LIN {X 0,Y 386.268,Z 340.052,A -85,B 0,C 180,E1 13716.91,E2 13716.91} C_VEL
LIN {X 0,Y 373.935,Z 326.395,A -85,B 0,C 180,E1 13713.839,E2 13713.839} C_VEL
LIN {X 0,Y 356.934,Z 301.733,A -85,B 0,C 180,E1 13708.485,E2 13708.485} C_VEL
LIN {X 0,Y 348.808,Z 290.548,A -85,B 0,C 180,E1 13705.376,E2 13705.376} C_VEL
LIN {X 0,Y 345.384,Z 285.946,A -85,B 0,C 180,E1 13703.91,E2 13703.91} C_VEL
LIN {X 0,Y 341.987,Z 281.466,A -85,B 0,C 180,E1 13702.339,E2 13702.339} C_VEL
LIN {X 0,Y 338.204,Z 276.56,A -85,B 0,C 180,E1 13700.418,E2 13700.418} C_VEL
LIN {X 0,Y 334.673,Z 272.149,A -85,B 0,C 180,E1 13698.418,E2 13698.418} C_VEL
LIN {X 0,Y 333.52,Z 270.824,A -85,B 0,C 180,E1 13697.716,E2 13697.716} C_VEL
LIN {X 0,Y 330.176,Z 266.785,A -85,B 0,C 180,E1 13695.456,E2 13695.456} C_VEL
LIN {X 0,Y 329.315,Z 265.342,A -85,B 0,C 180,E1 13694.776,E2 13694.776} C_VEL
LIN {X 0,Y 326.007,Z 262.321,A -85,B 0,C 180,E1 13692.038,E2 13692.038} C_VEL
LIN {X 0,Y 324.468,Z 259.24,A -85,B 0,C 180,E1 13690.296,E2 13690.296} C_VEL
LIN {X 0,Y 319.963,Z 254.972,A -85,B 0,C 180,E1 13681.074,E2 13681.074} C_VEL
LIN {X 0,Y 320.128,Z 255.393,A -85,B 0,C 180,E1 13677.852,E2 13677.852} C_VEL
LIN {X 0,Y 324.571,Z 259.436,A -85,B 0,C 180,E1 13669.886,E2 13669.886} C_VEL
LIN {X 0,Y 326.879,Z 263.417,A -85,B 0,C 180,E1 13667.456,E2 13667.456} C_VEL
LIN {X 0,Y 329.69,Z 265.855,A -85,B 0,C 180,E1 13665.241,E2 13665.241} C_VEL
LIN {X 0,Y 332.506,Z 269.885,A -85,B 0,C 180,E1 13663.221,E2 13663.221} C_VEL
LIN {X 0,Y 334.533,Z 271.893,A -85,B 0,C 180,E1 13661.98,E2 13661.98} C_VEL
LIN {X 0,Y 337.954,Z 276.34,A -85,B 0,C 180,E1 13660.018,E2 13660.018} C_VEL
LIN {X 0,Y 339.714,Z 278.629,A -85,B 0,C 180,E1 13659.091,E2 13659.091} C_VEL
LIN {X 0,Y 343.732,Z 283.696,A -85,B 0,C 180,E1 13657.148,E2 13657.148} C_VEL
LIN {X 0,Y 348.055,Z 289.495,A -85,B 0,C 180,E1 13655.247,E2 13655.247} C_VEL
LIN {X 0,Y 354.37,Z 298.173,A -85,B 0,C 180,E1 13652.754,E2 13652.754} C_VEL
LIN {X 0,Y 356.73,Z 301.564,A -85,B 0,C 180,E1 13651.89,E2 13651.89} C_VEL
LIN {X 0,Y 358.866,Z 306.87,A -85,B 0,C 180,E1 13651.048,E2 13651.048} C_VEL
LIN {X 0,Y 363.911,Z 325.647,A -85,B 0,C 180,E1 13648.944,E2 13648.944} C_VEL
LIN {X 0,Y 365.246,Z 328.766,A -85,B 0,C 180,E1 13648.485,E2 13648.485} C_VEL
LIN {X 0,Y 373.121,Z 344.861,A -85,B 0,C 180,E1 13646.031,E2 13646.031} C_VEL
LIN {X 0,Y 375.226,Z 349.974,A -85,B 0,C 180,E1 13645.391,E2 13645.391} C_VEL
LIN {X 0,Y 363.631,Z 518.512,A -85,B 0,C 180,E1 13642.347,E2 13642.347} C_VEL
LIN {X 0,Y 361.378,Z 537.609,A -85,B 0,C 180,E1 13641.872,E2 13641.872} C_VEL
LIN {X 0,Y 357.513,Z 560.275,A -85,B 0,C 180,E1 13641.106,E2 13641.106} C_VEL
LIN {X 0,Y 353.084,Z 580.15,A -85,B 0,C 180,E1 13640.185,E2 13640.185} C_VEL
LIN {X 0,Y 348.65,Z 597.084,A -85,B 0,C 180,E1 13639.202,E2 13639.202} C_VEL
LIN {X 0,Y 343.899,Z 612.945,A -85,B 0,C 180,E1 13638.092,E2 13638.092} C_VEL
LIN {X 0,Y 338.731,Z 628.386,A -85,B 0,C 180,E1 13636.804,E2 13636.804} C_VEL
LIN {X 0,Y 333.209,Z 643.365,A -85,B 0,C 180,E1 13635.324,E2 13635.324} C_VEL
LIN {X 0,Y 326.894,Z 659.095,A -85,B 0,C 180,E1 13633.482,E2 13633.482} C_VEL
LIN {X 0,Y 318.806,Z 677.555,A -85,B 0,C 180,E1 13630.832,E2 13630.832} C_VEL
LIN {X 0,Y 312.71,Z 690.554,A -85,B 0,C 180,E1 13628.567,E2 13628.567} C_VEL
LIN {X 0,Y 306.921,Z 702.441,A -85,B 0,C 180,E1 13626.127,E2 13626.127} C_VEL
LIN {X 0,Y 301.69,Z 712.936,A -85,B 0,C 180,E1 13623.601,E2 13623.601} C_VEL
LIN {X 0,Y 296.723,Z 722.827,A -85,B 0,C 180,E1 13620.806,E2 13620.806} C_VEL
LIN {X 0,Y 292.163,Z 732.011,A -85,B 0,C 180,E1 13617.735,E2 13617.735} C_VEL
LIN {X 0,Y 287.756,Z 741.331,A -85,B 0,C 180,E1 13613.985,E2 13613.985} C_VEL
LIN {X 0,Y 283.988,Z 749.983,A -85,B 0,C 180,E1 13609.538,E2 13609.538} C_VEL
LIN {X 0,Y 281.915,Z 755.6,A -85,B 0,C 180,E1 13605.847,E2 13605.847} C_VEL
LIN {X 0,Y 280.717,Z 759.775,A -85,B 0,C 180,E1 13602.338,E2 13602.338} C_VEL
LIN {X 0,Y 280.122,Z 762.882,A -85,B 0,C 180,E1 13598.828,E2 13598.828} C_VEL
LIN {X 0,Y 279.95,Z 764.861,A -85,B 0,C 180,E1 13595.533,E2 13595.533} C_VEL
LIN {X 0,Y 279.965,Z 765.937,A -85,B 0,C 180,E1 13592.251,E2 13592.251} C_VEL
LIN {X 0,Y 279.98,Z 766.115,A -85,B 0,C 180,E1 13588.977,E2 13588.977} C_VEL
LIN {X 0,Y 279.944,Z 765.306,A -85,B 0,C 180,E1 13585.494,E2 13585.494} C_VEL
LIN {X 0,Y 280.051,Z 763.477,A -85,B 0,C 180,E1 13581.997,E2 13581.997} C_VEL
LIN {X 0,Y 280.571,Z 760.402,A -85,B 0,C 180,E1 13578.281,E2 13578.281} C_VEL
LIN {X 0,Y 281.653,Z 756.413,A -85,B 0,C 180,E1 13574.771,E2 13574.771} C_VEL
LIN {X 0,Y 283.447,Z 751.32,A -85,B 0,C 180,E1 13571.279,E2 13571.279} C_VEL
LIN {X 0,Y 286.041,Z 745.066,A -85,B 0,C 180,E1 13567.823,E2 13567.823} C_VEL
LIN {X 0,Y 289.479,Z 737.579,A -85,B 0,C 180,E1 13564.424,E2 13564.424} C_VEL
LIN {X 0,Y 294.639,Z 727.132,A -85,B 0,C 180,E1 13560.528,E2 13560.528} C_VEL
LIN {X 0,Y 300.694,Z 714.948,A -85,B 0,C 180,E1 13556.927,E2 13556.927} C_VEL
LIN {X 0,Y 306.139,Z 704.024,A -85,B 0,C 180,E1 13554.228,E2 13554.228} C_VEL
LIN {X 0,Y 311.866,Z 692.294,A -85,B 0,C 180,E1 13551.768,E2 13551.768} C_VEL
LIN {X 0,Y 317.867,Z 679.553,A -85,B 0,C 180,E1 13549.497,E2 13549.497} C_VEL
LIN {X 0,Y 324.119,Z 665.583,A -85,B 0,C 180,E1 13547.386,E2 13547.386} C_VEL
LIN {X 0,Y 331.869,Z 646.919,A -85,B 0,C 180,E1 13545.055,E2 13545.055} C_VEL
LIN {X 0,Y 338.168,Z 629.997,A -85,B 0,C 180,E1 13543.342,E2 13543.342} C_VEL
LIN {X 0,Y 343.312,Z 614.785,A -85,B 0,C 180,E1 13542.048,E2 13542.048} C_VEL
LIN {X 0,Y 348.21,Z 598.635,A -85,B 0,C 180,E1 13540.898,E2 13540.898} C_VEL
LIN {X 0,Y 352.296,Z 583.32,A -85,B 0,C 180,E1 13539.985,E2 13539.985} C_VEL
LIN {X 0,Y 356.088,Z 566.94,A -85,B 0,C 180,E1 13539.183,E2 13539.183} C_VEL
LIN {X 0,Y 359.407,Z 549.856,A -85,B 0,C 180,E1 13538.516,E2 13538.516} C_VEL
LIN {X 0,Y 362.097,Z 532.301,A -85,B 0,C 180,E1 13537.984,E2 13537.984} C_VEL
LIN {X 0,Y 364.159,Z 512.509,A -85,B 0,C 180,E1 13537.527,E2 13537.527} C_VEL
LIN {X 0,Y 375.197,Z 349.477,A -85,B 0,C 180,E1 13534.586,E2 13534.586} C_VEL
LIN {X 0,Y 367.633,Z 333.537,A -85,B 0,C 180,E1 13532.283,E2 13532.283} C_VEL
LIN {X 0,Y 360.351,Z 319.565,A -85,B 0,C 180,E1 13529.873,E2 13529.873} C_VEL
LIN {X 0,Y 353.374,Z 307.386,A -85,B 0,C 180,E1 13527.332,E2 13527.332} C_VEL
LIN {X 0,Y 346.425,Z 297.518,A -85,B 0,C 180,E1 13524.559,E2 13524.559} C_VEL
LIN {X 0,Y 342.821,Z 292.619,A -85,B 0,C 180,E1 13522.961,E2 13522.961} C_VEL
LIN {X 0,Y 339.925,Z 288.734,A -85,B 0,C 180,E1 13521.573,E2 13521.573} C_VEL
LIN {X 0,Y 336.229,Z 283.884,A -85,B 0,C 180,E1 13519.636,E2 13519.636} C_VEL
LIN {X 0,Y 332.684,Z 279.147,A -85,B 0,C 180,E1 13517.536,E2 13517.536} C_VEL
LIN {X 0,Y 328.89,Z 274.782,A -85,B 0,C 180,E1 13514.976,E2 13514.976} C_VEL
LIN {X 0,Y 327.794,Z 273.016,A -85,B 0,C 180,E1 13514.098,E2 13514.098} C_VEL
LIN {X 0,Y 324.631,Z 269.906,A -85,B 0,C 180,E1 13511.369,E2 13511.369} C_VEL
LIN {X 0,Y 323.127,Z 267.059,A -85,B 0,C 180,E1 13509.619,E2 13509.619} C_VEL
LIN {X 0,Y 318.996,Z 262.945,A -85,B 0,C 180,E1 13500.898,E2 13500.898} C_VEL
LIN {X 0,Y 319.101,Z 263.237,A -85,B 0,C 180,E1 13497.845,E2 13497.845} C_VEL
LIN {X 0,Y 323.392,Z 267.413,A -85,B 0,C 180,E1 13489.759,E2 13489.759} C_VEL
LIN {X 0,Y 325.671,Z 271.291,A -85,B 0,C 180,E1 13487.319,E2 13487.319} C_VEL
LIN {X 0,Y 328.214,Z 273.554,A -85,B 0,C 180,E1 13485.263,E2 13485.263} C_VEL
LIN {X 0,Y 331.228,Z 277.785,A -85,B 0,C 180,E1 13483.064,E2 13483.064} C_VEL
LIN {X 0,Y 332.948,Z 279.629,A -85,B 0,C 180,E1 13481.981,E2 13481.981} C_VEL
LIN {X 0,Y 336.629,Z 284.252,A -85,B 0,C 180,E1 13479.845,E2 13479.845} C_VEL
LIN {X 0,Y 341.914,Z 291.371,A -85,B 0,C 180,E1 13477.157,E2 13477.157} C_VEL
LIN {X 0,Y 346.173,Z 297.193,A -85,B 0,C 180,E1 13475.24,E2 13475.24} C_VEL
LIN {X 0,Y 352.796,Z 306.559,A -85,B 0,C 180,E1 13472.577,E2 13472.577} C_VEL
LIN {X 0,Y 360.002,Z 317.337,A -85,B 0,C 180,E1 13470.004,E2 13470.004} C_VEL
LIN {X 0,Y 371.633,Z 334.055,A -85,B 0,C 180,E1 13466.433,E2 13466.433} C_VEL
LIN {X 0,Y 387.013,Z 350.884,A -85,B 0,C 180,E1 13462.616,E2 13462.616} C_VEL
LIN {X 0,Y 404.416,Z 365.915,A -85,B 0,C 180,E1 13459.019,E2 13459.019} C_VEL
LIN {X 0,Y 413.951,Z 373.978,A -85,B 0,C 180,E1 13456.97,E2 13456.97} C_VEL
LIN {X 0,Y 423.451,Z 382.101,A -85,B 0,C 180,E1 13454.752,E2 13454.752} C_VEL
LIN {X 0,Y 431.998,Z 389.621,A -85,B 0,C 180,E1 13452.556,E2 13452.556} C_VEL
LIN {X 0,Y 441.62,Z 398.394,A -85,B 0,C 180,E1 13449.815,E2 13449.815} C_VEL
LIN {X 0,Y 450.481,Z 406.222,A -85,B 0,C 180,E1 13447.171,E2 13447.171} C_VEL
LIN {X 0,Y 459.526,Z 414.01,A -85,B 0,C 180,E1 13444.334,E2 13444.334} C_VEL
LIN {X 0,Y 466.257,Z 419.625,A -85,B 0,C 180,E1 13442.104,E2 13442.104} C_VEL
LIN {X 0,Y 473.318,Z 425.906,A -85,B 0,C 180,E1 13439.621,E2 13439.621} C_VEL
LIN {X 0,Y 478.445,Z 429.943,A -85,B 0,C 180,E1 13437.74,E2 13437.74} C_VEL
LIN {X 0,Y 484.241,Z 434.888,A -85,B 0,C 180,E1 13435.432,E2 13435.432} C_VEL
LIN {X 0,Y 488.516,Z 438.069,A -85,B 0,C 180,E1 13433.648,E2 13433.648} C_VEL
LIN {X 0,Y 493.363,Z 442.438,A -85,B 0,C 180,E1 13431.392,E2 13431.392} C_VEL
LIN {X 0,Y 498.263,Z 445.648,A -85,B 0,C 180,E1 13428.969,E2 13428.969} C_VEL
LIN {X 0,Y 502.59,Z 449.801,A -85,B 0,C 180,E1 13426.478,E2 13426.478} C_VEL
LIN {X 0,Y 506.276,Z 452.541,A -85,B 0,C 180,E1 13424.057,E2 13424.057} C_VEL
LIN {X 0,Y 509.659,Z 454.3,A -85,B 0,C 180,E1 13421.542,E2 13421.542} C_VEL
LIN {X 0,Y 510.793,Z 455.335,A -85,B 0,C 180,E1 13420.488,E2 13420.488} C_VEL
LIN {X 0,Y 513.093,Z 457.868,A -85,B 0,C 180,E1 13417.952,E2 13417.952} C_VEL
LIN {X 0,Y 514.62,Z 459.31,A -85,B 0,C 180,E1 13415.686,E2 13415.686} C_VEL
LIN {X 0,Y 515.845,Z 460.261,A -85,B 0,C 180,E1 13413,E2 13413} C_VEL
LIN {X 0,Y 516.274,Z 460.529,A -85,B 0,C 180,E1 13410.555,E2 13410.555} C_VEL
LIN {X 0,Y 516.046,Z 460.366,A -85,B 0,C 180,E1 13407.779,E2 13407.779} C_VEL
LIN {X 0,Y 515.181,Z 459.728,A -85,B 0,C 180,E1 13405.325,E2 13405.325} C_VEL
LIN {X 0,Y 513.6,Z 458.417,A -85,B 0,C 180,E1 13402.731,E2 13402.731} C_VEL
LIN {X 0,Y 511.457,Z 456.139,A -85,B 0,C 180,E1 13400.169,E2 13400.169} C_VEL
LIN {X 0,Y 509.789,Z 454.349,A -85,B 0,C 180,E1 13398.576,E2 13398.576} C_VEL
LIN {X 0,Y 506.453,Z 452.644,A -85,B 0,C 180,E1 13396.064,E2 13396.064} C_VEL
LIN {X 0,Y 502.909,Z 450.074,A -85,B 0,C 180,E1 13393.722,E2 13393.722} C_VEL
LIN {X 0,Y 498.849,Z 446.206,A -85,B 0,C 180,E1 13391.358,E2 13391.358} C_VEL
LIN {X 0,Y 493.606,Z 442.619,A -85,B 0,C 180,E1 13388.72,E2 13388.72} C_VEL
LIN {X 0,Y 488.817,Z 438.383,A -85,B 0,C 180,E1 13386.495,E2 13386.495} C_VEL
LIN {X 0,Y 485.363,Z 435.679,A -85,B 0,C 180,E1 13385.018,E2 13385.018} C_VEL
LIN {X 0,Y 479.539,Z 431.003,A -85,B 0,C 180,E1 13382.699,E2 13382.699} C_VEL
LIN {X 0,Y 475.675,Z 427.655,A -85,B 0,C 180,E1 13381.23,E2 13381.23} C_VEL
LIN {X 0,Y 469.252,Z 422.415,A -85,B 0,C 180,E1 13378.936,E2 13378.936} C_VEL
LIN {X 0,Y 464.33,Z 418.154,A -85,B 0,C 180,E1 13377.248,E2 13377.248} C_VEL
LIN {X 0,Y 456.023,Z 410.909,A -85,B 0,C 180,E1 13374.544,E2 13374.544} C_VEL
LIN {X 0,Y 448.696,Z 404.527,A -85,B 0,C 180,E1 13372.288,E2 13372.288} C_VEL
LIN {X 0,Y 440.156,Z 396.98,A -85,B 0,C 180,E1 13369.755,E2 13369.755} C_VEL
LIN {X 0,Y 431.296,Z 388.943,A -85,B 0,C 180,E1 13367.251,E2 13367.251} C_VEL
LIN {X 0,Y 421.982,Z 380.697,A -85,B 0,C 180,E1 13364.872,E2 13364.872} C_VEL
LIN {X 0,Y 413.139,Z 373.258,A -85,B 0,C 180,E1 13362.85,E2 13362.85} C_VEL
LIN {X 0,Y 403.162,Z 364.77,A -85,B 0,C 180,E1 13360.713,E2 13360.713} C_VEL
LIN {X 0,Y 385.913,Z 349.796,A -85,B 0,C 180,E1 13357.135,E2 13357.135} C_VEL
LIN {X 0,Y 371.026,Z 333.282,A -85,B 0,C 180,E1 13353.397,E2 13353.397} C_VEL
LIN {X 0,Y 359.686,Z 316.803,A -85,B 0,C 180,E1 13349.887,E2 13349.887} C_VEL
LIN {X 0,Y 351.241,Z 304.196,A -85,B 0,C 180,E1 13346.821,E2 13346.821} C_VEL
LIN {X 0,Y 343.795,Z 293.837,A -85,B 0,C 180,E1 13343.709,E2 13343.709} C_VEL
LIN {X 0,Y 339.862,Z 288.649,A -85,B 0,C 180,E1 13341.849,E2 13341.849} C_VEL
LIN {X 0,Y 336.322,Z 283.967,A -85,B 0,C 180,E1 13339.993,E2 13339.993} C_VEL
LIN {X 0,Y 332.758,Z 279.293,A -85,B 0,C 180,E1 13337.893,E2 13337.893} C_VEL
LIN {X 0,Y 328.737,Z 274.526,A -85,B 0,C 180,E1 13335.164,E2 13335.164} C_VEL
LIN {X 0,Y 327.895,Z 273.084,A -85,B 0,C 180,E1 13334.481,E2 13334.481} C_VEL
LIN {X 0,Y 324.677,Z 270.01,A -85,B 0,C 180,E1 13331.727,E2 13331.727} C_VEL
LIN {X 0,Y 323.175,Z 267.07,A -85,B 0,C 180,E1 13329.978,E2 13329.978} C_VEL
LIN {X 0,Y 318.987,Z 262.924,A -85,B 0,C 180,E1 13321.078,E2 13321.078} C_VEL
LIN {X 0,Y 319.12,Z 263.29,A -85,B 0,C 180,E1 13318.025,E2 13318.025} C_VEL
LIN {X 0,Y 323.351,Z 267.336,A -85,B 0,C 180,E1 13310.118,E2 13310.118} C_VEL
LIN {X 0,Y 325.712,Z 271.322,A -85,B 0,C 180,E1 13307.591,E2 13307.591} C_VEL
LIN {X 0,Y 328.256,Z 273.631,A -85,B 0,C 180,E1 13305.536,E2 13305.536} C_VEL
LIN {X 0,Y 331.282,Z 277.826,A -85,B 0,C 180,E1 13303.337,E2 13303.337} C_VEL
LIN {X 0,Y 332.936,Z 279.602,A -85,B 0,C 180,E1 13302.297,E2 13302.297} C_VEL
LIN {X 0,Y 336.535,Z 284.175,A -85,B 0,C 180,E1 13300.202,E2 13300.202} C_VEL
LIN {X 0,Y 341.897,Z 291.332,A -85,B 0,C 180,E1 13297.473,E2 13297.473} C_VEL
LIN {X 0,Y 346.064,Z 297.019,A -85,B 0,C 180,E1 13295.595,E2 13295.595} C_VEL
LIN {X 0,Y 352.278,Z 305.799,A -85,B 0,C 180,E1 13293.082,E2 13293.082} C_VEL
LIN {X 0,Y 355.942,Z 311.724,A -85,B 0,C 180,E1 13291.703,E2 13291.703} C_VEL
LIN {X 0,Y 362.038,Z 322.693,A -85,B 0,C 180,E1 13289.549,E2 13289.549} C_VEL
LIN {X 0,Y 365.246,Z 328.766,A -85,B 0,C 180,E1 13288.485,E2 13288.485} C_VEL
LIN {X 0,Y 366.5,Z 332.86,A -85,B 0,C 180,E1 13288.021,E2 13288.021} C_VEL
LIN {X 0,Y 368.162,Z 346.842,A -85,B 0,C 180,E1 13287.118,E2 13287.118} C_VEL
LIN {X 0,Y 369.102,Z 349.82,A -85,B 0,C 180,E1 13286.791,E2 13286.791} C_VEL
LIN {X 0,Y 370.477,Z 353.325,A -85,B 0,C 180,E1 13286.35,E2 13286.35} C_VEL
LIN {X 0,Y 358.789,Z 518.345,A -85,B 0,C 180,E1 13283.361,E2 13283.361} C_VEL
LIN {X 0,Y 356.461,Z 537.596,A -85,B 0,C 180,E1 13282.882,E2 13282.882} C_VEL
LIN {X 0,Y 352.312,Z 561.069,A -85,B 0,C 180,E1 13282.081,E2 13282.081} C_VEL
LIN {X 0,Y 347.999,Z 579.939,A -85,B 0,C 180,E1 13281.203,E2 13281.203} C_VEL
LIN {X 0,Y 343.442,Z 596.908,A -85,B 0,C 180,E1 13280.219,E2 13280.219} C_VEL
LIN {X 0,Y 338.565,Z 612.769,A -85,B 0,C 180,E1 13279.108,E2 13279.108} C_VEL
LIN {X 0,Y 333.249,Z 628.209,A -85,B 0,C 180,E1 13277.817,E2 13277.817} C_VEL
LIN {X 0,Y 327.566,Z 643.188,A -85,B 0,C 180,E1 13276.331,E2 13276.331} C_VEL
LIN {X 0,Y 321.054,Z 658.917,A -85,B 0,C 180,E1 13274.479,E2 13274.479} C_VEL
LIN {X 0,Y 312.923,Z 676.917,A -85,B 0,C 180,E1 13271.882,E2 13271.882} C_VEL
LIN {X 0,Y 306.383,Z 690.376,A -85,B 0,C 180,E1 13269.516,E2 13269.516} C_VEL
LIN {X 0,Y 300.369,Z 702.263,A -85,B 0,C 180,E1 13267.045,E2 13267.045} C_VEL
LIN {X 0,Y 294.917,Z 712.758,A -85,B 0,C 180,E1 13264.48,E2 13264.48} C_VEL
LIN {X 0,Y 289.728,Z 722.649,A -85,B 0,C 180,E1 13261.635,E2 13261.635} C_VEL
LIN {X 0,Y 284.949,Z 731.833,A -85,B 0,C 180,E1 13258.5,E2 13258.5} C_VEL
LIN {X 0,Y 280.306,Z 741.152,A -85,B 0,C 180,E1 13254.664,E2 13254.664} C_VEL
LIN {X 0,Y 276.312,Z 749.804,A -85,B 0,C 180,E1 13250.104,E2 13250.104} C_VEL
LIN {X 0,Y 274.095,Z 755.423,A -85,B 0,C 180,E1 13246.311,E2 13246.311} C_VEL
LIN {X 0,Y 272.799,Z 759.597,A -85,B 0,C 180,E1 13242.702,E2 13242.702} C_VEL
LIN {X 0,Y 272.148,Z 762.705,A -85,B 0,C 180,E1 13239.089,E2 13239.089} C_VEL
LIN {X 0,Y 271.955,Z 764.686,A -85,B 0,C 180,E1 13235.696,E2 13235.696} C_VEL
LIN {X 0,Y 271.965,Z 765.762,A -85,B 0,C 180,E1 13232.317,E2 13232.317} C_VEL
LIN {X 0,Y 271.981,Z 765.94,A -85,B 0,C 180,E1 13228.947,E2 13228.947} C_VEL
LIN {X 0,Y 271.944,Z 765.131,A -85,B 0,C 180,E1 13225.361,E2 13225.361} C_VEL
LIN {X 0,Y 272.082,Z 763.152,A -85,B 0,C 180,E1 13221.548,E2 13221.548} C_VEL
LIN {X 0,Y 272.642,Z 760.225,A -85,B 0,C 180,E1 13217.935,E2 13217.935} C_VEL
LIN {X 0,Y 273.813,Z 756.235,A -85,B 0,C 180,E1 13214.324,E2 13214.324} C_VEL
LIN {X 0,Y 275.735,Z 751.141,A -85,B 0,C 180,E1 13210.735,E2 13210.735} C_VEL
LIN {X 0,Y 278.49,Z 744.888,A -85,B 0,C 180,E1 13207.188,E2 13207.188} C_VEL
LIN {X 0,Y 282.123,Z 737.4,A -85,B 0,C 180,E1 13203.707,E2 13203.707} C_VEL
LIN {X 0,Y 287.548,Z 726.954,A -85,B 0,C 180,E1 13199.726,E2 13199.726} C_VEL
LIN {X 0,Y 293.83,Z 714.862,A -85,B 0,C 180,E1 13196.082,E2 13196.082} C_VEL
LIN {X 0,Y 299.554,Z 703.846,A -85,B 0,C 180,E1 13193.316,E2 13193.316} C_VEL
LIN {X 0,Y 305.486,Z 692.155,A -85,B 0,C 180,E1 13190.83,E2 13190.83} C_VEL
LIN {X 0,Y 311.725,Z 679.375,A -85,B 0,C 180,E1 13188.526,E2 13188.526} C_VEL
LIN {X 0,Y 318.191,Z 665.406,A -85,B 0,C 180,E1 13186.396,E2 13186.396} C_VEL
LIN {X 0,Y 326.187,Z 646.742,A -85,B 0,C 180,E1 13184.05,E2 13184.05} C_VEL
LIN {X 0,Y 332.77,Z 629.544,A -85,B 0,C 180,E1 13182.304,E2 13182.304} C_VEL
LIN {X 0,Y 338.263,Z 613.689,A -85,B 0,C 180,E1 13180.962,E2 13180.962} C_VEL
LIN {X 0,Y 343.101,Z 598.075,A -85,B 0,C 180,E1 13179.856,E2 13179.856} C_VEL
LIN {X 0,Y 347.497,Z 581.901,A -85,B 0,C 180,E1 13178.901,E2 13178.901} C_VEL
LIN {X 0,Y 351.332,Z 565.526,A -85,B 0,C 180,E1 13178.112,E2 13178.112} C_VEL
LIN {X 0,Y 354.815,Z 547.736,A -85,B 0,C 180,E1 13177.434,E2 13177.434} C_VEL
LIN {X 0,Y 358.133,Z 525.425,A -85,B 0,C 180,E1 13176.79,E2 13176.79} C_VEL
LIN {X 0,Y 360.831,Z 491.406,A -85,B 0,C 180,E1 13176.123,E2 13176.123} C_VEL
LIN {X 0,Y 370.425,Z 352.817,A -85,B 0,C 180,E1 13173.621,E2 13173.621} C_VEL
LIN {X 0,Y 363.461,Z 337.977,A -85,B 0,C 180,E1 13171.398,E2 13171.398} C_VEL
LIN {X 0,Y 355.897,Z 323.266,A -85,B 0,C 180,E1 13168.759,E2 13168.759} C_VEL
LIN {X 0,Y 350.2,Z 313.406,A -85,B 0,C 180,E1 13166.587,E2 13166.587} C_VEL
LIN {X 0,Y 343.823,Z 304.159,A -85,B 0,C 180,E1 13163.934,E2 13163.934} C_VEL
LIN {X 0,Y 338.469,Z 296.639,A -85,B 0,C 180,E1 13161.398,E2 13161.398} C_VEL
LIN {X 0,Y 334.22,Z 291.13,A -85,B 0,C 180,E1 13159.123,E2 13159.123} C_VEL
LIN {X 0,Y 330.453,Z 286.11,A -85,B 0,C 180,E1 13156.796,E2 13156.796} C_VEL
LIN {X 0,Y 327.14,Z 281.961,A -85,B 0,C 180,E1 13154.424,E2 13154.424} C_VEL
LIN {X 0,Y 326.197,Z 280.616,A -85,B 0,C 180,E1 13153.652,E2 13153.652} C_VEL
LIN {X 0,Y 323.15,Z 277.325,A -85,B 0,C 180,E1 13150.88,E2 13150.88} C_VEL
LIN {X 0,Y 321.846,Z 274.873,A -85,B 0,C 180,E1 13149.297,E2 13149.297} C_VEL
LIN {X 0,Y 318.008,Z 270.854,A -85,B 0,C 180,E1 13140.721,E2 13140.721} C_VEL
LIN {X 0,Y 318.154,Z 271.253,A -85,B 0,C 180,E1 13137.659,E2 13137.659} C_VEL
LIN {X 0,Y 322.179,Z 275.301,A -85,B 0,C 180,E1 13129.991,E2 13129.991} C_VEL
LIN {X 0,Y 324.508,Z 279.194,A -85,B 0,C 180,E1 13127.454,E2 13127.454} C_VEL
LIN {X 0,Y 326.793,Z 281.317,A -85,B 0,C 180,E1 13125.56,E2 13125.56} C_VEL
LIN {X 0,Y 330.007,Z 285.727,A -85,B 0,C 180,E1 13123.181,E2 13123.181} C_VEL
LIN {X 0,Y 331.427,Z 287.428,A -85,B 0,C 180,E1 13122.259,E2 13122.259} C_VEL
LIN {X 0,Y 335.791,Z 293.151,A -85,B 0,C 180,E1 13119.694,E2 13119.694} C_VEL
LIN {X 0,Y 339.93,Z 298.753,A -85,B 0,C 180,E1 13117.564,E2 13117.564} C_VEL
LIN {X 0,Y 345.555,Z 306.5,A -85,B 0,C 180,E1 13115.01,E2 13115.01} C_VEL
LIN {X 0,Y 354.41,Z 319.625,A -85,B 0,C 180,E1 13111.524,E2 13111.524} C_VEL
LIN {X 0,Y 368.498,Z 340.631,A -85,B 0,C 180,E1 13106.948,E2 13106.948} C_VEL
LIN {X 0,Y 383.658,Z 357.495,A -85,B 0,C 180,E1 13103.078,E2 13103.078} C_VEL
LIN {X 0,Y 403.445,Z 374.675,A -85,B 0,C 180,E1 13098.946,E2 13098.946} C_VEL
LIN {X 0,Y 411.876,Z 381.715,A -85,B 0,C 180,E1 13097.143,E2 13097.143} C_VEL
LIN {X 0,Y 421.313,Z 389.639,A -85,B 0,C 180,E1 13094.989,E2 13094.989} C_VEL
LIN {X 0,Y 429.934,Z 397.176,A -85,B 0,C 180,E1 13092.788,E2 13092.788} C_VEL
LIN {X 0,Y 438.951,Z 405.269,A -85,B 0,C 180,E1 13090.262,E2 13090.262} C_VEL
LIN {X 0,Y 448.23,Z 413.453,A -85,B 0,C 180,E1 13087.511,E2 13087.511} C_VEL
LIN {X 0,Y 457.07,Z 420.986,A -85,B 0,C 180,E1 13084.77,E2 13084.77} C_VEL
LIN {X 0,Y 464.208,Z 427.004,A -85,B 0,C 180,E1 13082.43,E2 13082.43} C_VEL
LIN {X 0,Y 471.575,Z 433.471,A -85,B 0,C 180,E1 13079.863,E2 13079.863} C_VEL
LIN {X 0,Y 476.902,Z 437.655,A -85,B 0,C 180,E1 13077.919,E2 13077.919} C_VEL
LIN {X 0,Y 482.84,Z 442.669,A -85,B 0,C 180,E1 13075.576,E2 13075.576} C_VEL
LIN {X 0,Y 487.337,Z 446.052,A -85,B 0,C 180,E1 13073.709,E2 13073.709} C_VEL
LIN {X 0,Y 492.23,Z 450.378,A -85,B 0,C 180,E1 13071.444,E2 13071.444} C_VEL
LIN {X 0,Y 497.637,Z 454.079,A -85,B 0,C 180,E1 13068.75,E2 13068.75} C_VEL
LIN {X 0,Y 501.65,Z 457.858,A -85,B 0,C 180,E1 13066.439,E2 13066.439} C_VEL
LIN {X 0,Y 505.24,Z 460.477,A -85,B 0,C 180,E1 13064.087,E2 13064.087} C_VEL
LIN {X 0,Y 508.651,Z 462.234,A -85,B 0,C 180,E1 13061.565,E2 13061.565} C_VEL
LIN {X 0,Y 509.906,Z 463.464,A -85,B 0,C 180,E1 13060.392,E2 13060.392} C_VEL
LIN {X 0,Y 512.177,Z 465.921,A -85,B 0,C 180,E1 13057.853,E2 13057.853} C_VEL
LIN {X 0,Y 513.706,Z 467.304,A -85,B 0,C 180,E1 13055.584,E2 13055.584} C_VEL
LIN {X 0,Y 514.89,Z 468.216,A -85,B 0,C 180,E1 13052.894,E2 13052.894} C_VEL
LIN {X 0,Y 515.314,Z 468.47,A -85,B 0,C 180,E1 13050.445,E2 13050.445} C_VEL
LIN {X 0,Y 515.067,Z 468.307,A -85,B 0,C 180,E1 13047.775,E2 13047.775} C_VEL
LIN {X 0,Y 514.243,Z 467.711,A -85,B 0,C 180,E1 13045.428,E2 13045.428} C_VEL
LIN {X 0,Y 512.605,Z 466.365,A -85,B 0,C 180,E1 13042.717,E2 13042.717} C_VEL
LIN {X 0,Y 510.459,Z 464.113,A -85,B 0,C 180,E1 13040.158,E2 13040.158} C_VEL
LIN {X 0,Y 508.78,Z 462.283,A -85,B 0,C 180,E1 13038.553,E2 13038.553} C_VEL
LIN {X 0,Y 505.417,Z 460.579,A -85,B 0,C 180,E1 13036.035,E2 13036.035} C_VEL
LIN {X 0,Y 501.851,Z 458.028,A -85,B 0,C 180,E1 13033.687,E2 13033.687} C_VEL
LIN {X 0,Y 497.753,Z 454.206,A -85,B 0,C 180,E1 13031.315,E2 13031.315} C_VEL
LIN {X 0,Y 492.529,Z 450.598,A -85,B 0,C 180,E1 13028.695,E2 13028.695} C_VEL
LIN {X 0,Y 487.641,Z 446.35,A -85,B 0,C 180,E1 13026.428,E2 13026.428} C_VEL
LIN {X 0,Y 484.306,Z 443.686,A -85,B 0,C 180,E1 13025.006,E2 13025.006} C_VEL
LIN {X 0,Y 478.388,Z 439.045,A -85,B 0,C 180,E1 13022.661,E2 13022.661} C_VEL
LIN {X 0,Y 473.956,Z 435.228,A -85,B 0,C 180,E1 13020.977,E2 13020.977} C_VEL
LIN {X 0,Y 467.477,Z 429.951,A -85,B 0,C 180,E1 13018.689,E2 13018.689} C_VEL
LIN {X 0,Y 461.873,Z 425.194,A -85,B 0,C 180,E1 13016.795,E2 13016.795} C_VEL
LIN {X 0,Y 453.321,Z 417.813,A -85,B 0,C 180,E1 13014.047,E2 13014.047} C_VEL
LIN {X 0,Y 446.033,Z 411.325,A -85,B 0,C 180,E1 13011.817,E2 13011.817} C_VEL
LIN {X 0,Y 438.152,Z 404.504,A -85,B 0,C 180,E1 13009.508,E2 13009.508} C_VEL
LIN {X 0,Y 429.304,Z 396.593,A -85,B 0,C 180,E1 13007.048,E2 13007.048} C_VEL
LIN {X 0,Y 419.866,Z 388.363,A -85,B 0,C 180,E1 13004.678,E2 13004.678} C_VEL
LIN {X 0,Y 411.376,Z 381.28,A -85,B 0,C 180,E1 13002.746,E2 13002.746} C_VEL
LIN {X 0,Y 401.592,Z 373.078,A -85,B 0,C 180,E1 13000.671,E2 13000.671} C_VEL
LIN {X 0,Y 382.303,Z 356.118,A -85,B 0,C 180,E1 12996.607,E2 12996.607} C_VEL
LIN {X 0,Y 367.9,Z 339.853,A -85,B 0,C 180,E1 12992.88,E2 12992.88} C_VEL
LIN {X 0,Y 351.607,Z 315.368,A -85,B 0,C 180,E1 12987.432,E2 12987.432} C_VEL
LIN {X 0,Y 343.843,Z 304.211,A -85,B 0,C 180,E1 12984.252,E2 12984.252} C_VEL
LIN {X 0,Y 338.408,Z 296.559,A -85,B 0,C 180,E1 12981.675,E2 12981.675} C_VEL
LIN {X 0,Y 334.311,Z 291.217,A -85,B 0,C 180,E1 12979.48,E2 12979.48} C_VEL
LIN {X 0,Y 330.398,Z 286.089,A -85,B 0,C 180,E1 12977.071,E2 12977.071} C_VEL
LIN {X 0,Y 326.995,Z 281.702,A -85,B 0,C 180,E1 12974.612,E2 12974.612} C_VEL
LIN {X 0,Y 326.262,Z 280.671,A -85,B 0,C 180,E1 12974.011,E2 12974.011} C_VEL
LIN {X 0,Y 323.194,Z 277.434,A -85,B 0,C 180,E1 12971.239,E2 12971.239} C_VEL
LIN {X 0,Y 321.892,Z 274.896,A -85,B 0,C 180,E1 12969.656,E2 12969.656} C_VEL
LIN {X 0,Y 318.002,Z 270.826,A -85,B 0,C 180,E1 12960.901,E2 12960.901} C_VEL
LIN {X 0,Y 318.209,Z 271.374,A -85,B 0,C 180,E1 12957.659,E2 12957.659} C_VEL
LIN {X 0,Y 322.139,Z 275.22,A -85,B 0,C 180,E1 12950.351,E2 12950.351} C_VEL
LIN {X 0,Y 324.548,Z 279.224,A -85,B 0,C 180,E1 12947.726,E2 12947.726} C_VEL
LIN {X 0,Y 326.773,Z 281.271,A -85,B 0,C 180,E1 12945.885,E2 12945.885} C_VEL
LIN {X 0,Y 329.803,Z 285.514,A -85,B 0,C 180,E1 12943.623,E2 12943.623} C_VEL
LIN {X 0,Y 331.352,Z 287.293,A -85,B 0,C 180,E1 12942.618,E2 12942.618} C_VEL
LIN {X 0,Y 335.757,Z 293.139,A -85,B 0,C 180,E1 12940.018,E2 12940.018} C_VEL
LIN {X 0,Y 339.911,Z 298.713,A -85,B 0,C 180,E1 12937.881,E2 12937.881} C_VEL
LIN {X 0,Y 345.624,Z 306.575,A -85,B 0,C 180,E1 12935.289,E2 12935.289} C_VEL
LIN {X 0,Y 351.746,Z 315.892,A -85,B 0,C 180,E1 12932.809,E2 12932.809} C_VEL
LIN {X 0,Y 358.447,Z 328.069,A -85,B 0,C 180,E1 12930.321,E2 12930.321} C_VEL
LIN {X 0,Y 366.358,Z 343.88,A -85,B 0,C 180,E1 12927.66,E2 12927.66} C_VEL
LIN {X 0,Y 369.102,Z 349.82,A -85,B 0,C 180,E1 12926.791,E2 12926.791} C_VEL
LIN {X 0,Y 369.576,Z 352.536,A -85,B 0,C 180,E1 12926.586,E2 12926.586} C_VEL
LIN {X 0,Y 369.012,Z 357.168,A -85,B 0,C 180,E1 12926.558,E2 12926.558} C_VEL
LIN {X 0,Y 365.102,Z 370.077,A -85,B 0,C 180,E1 12927.035,E2 12927.035} C_VEL
LIN {X 0,Y 364.616,Z 373.344,A -85,B 0,C 180,E1 12927.037,E2 12927.037} C_VEL
LIN {X 0,Y 354.042,Z 518.375,A -85,B 0,C 180,E1 12924.398,E2 12924.398} C_VEL
LIN {X 0,Y 351.612,Z 537.907,A -85,B 0,C 180,E1 12923.91,E2 12923.91} C_VEL
LIN {X 0,Y 347.267,Z 561.637,A -85,B 0,C 180,E1 12923.094,E2 12923.094} C_VEL
LIN {X 0,Y 342.829,Z 580.482,A -85,B 0,C 180,E1 12922.212,E2 12922.212} C_VEL
LIN {X 0,Y 338.346,Z 596.732,A -85,B 0,C 180,E1 12921.267,E2 12921.267} C_VEL
LIN {X 0,Y 333.341,Z 612.593,A -85,B 0,C 180,E1 12920.156,E2 12920.156} C_VEL
LIN {X 0,Y 327.876,Z 628.033,A -85,B 0,C 180,E1 12918.864,E2 12918.864} C_VEL
LIN {X 0,Y 322.028,Z 643.011,A -85,B 0,C 180,E1 12917.373,E2 12917.373} C_VEL
LIN {X 0,Y 315.278,Z 658.825,A -85,B 0,C 180,E1 12915.501,E2 12915.501} C_VEL
LIN {X 0,Y 306.636,Z 677.295,A -85,B 0,C 180,E1 12912.803,E2 12912.803} C_VEL
LIN {X 0,Y 300.144,Z 690.198,A -85,B 0,C 180,E1 12910.506,E2 12910.506} C_VEL
LIN {X 0,Y 293.899,Z 702.085,A -85,B 0,C 180,E1 12908.003,E2 12908.003} C_VEL
LIN {X 0,Y 288.16,Z 712.689,A -85,B 0,C 180,E1 12905.37,E2 12905.37} C_VEL
LIN {X 0,Y 282.799,Z 722.47,A -85,B 0,C 180,E1 12902.504,E2 12902.504} C_VEL
LIN {X 0,Y 277.788,Z 731.654,A -85,B 0,C 180,E1 12899.305,E2 12899.305} C_VEL
LIN {X 0,Y 272.896,Z 740.974,A -85,B 0,C 180,E1 12895.381,E2 12895.381} C_VEL
LIN {X 0,Y 268.661,Z 749.626,A -85,B 0,C 180,E1 12890.703,E2 12890.703} C_VEL
LIN {X 0,Y 266.26,Z 755.321,A -85,B 0,C 180,E1 12886.742,E2 12886.742} C_VEL
LIN {X 0,Y 264.888,Z 759.42,A -85,B 0,C 180,E1 12883.088,E2 12883.088} C_VEL
LIN {X 0,Y 264.172,Z 762.529,A -85,B 0,C 180,E1 12879.365,E2 12879.365} C_VEL
LIN {X 0,Y 263.961,Z 764.51,A -85,B 0,C 180,E1 12875.869,E2 12875.869} C_VEL
LIN {X 0,Y 263.965,Z 765.587,A -85,B 0,C 180,E1 12872.388,E2 12872.388} C_VEL
LIN {X 0,Y 263.982,Z 765.765,A -85,B 0,C 180,E1 12868.915,E2 12868.915} C_VEL
LIN {X 0,Y 263.944,Z 764.9,A -85,B 0,C 180,E1 12865.084,E2 12865.084} C_VEL
LIN {X 0,Y 264.106,Z 762.975,A -85,B 0,C 180,E1 12861.291,E2 12861.291} C_VEL
LIN {X 0,Y 264.719,Z 760.048,A -85,B 0,C 180,E1 12857.569,E2 12857.569} C_VEL
LIN {X 0,Y 265.987,Z 756.057,A -85,B 0,C 180,E1 12853.851,E2 12853.851} C_VEL
LIN {X 0,Y 268.049,Z 750.963,A -85,B 0,C 180,E1 12850.159,E2 12850.159} C_VEL
LIN {X 0,Y 270.975,Z 744.709,A -85,B 0,C 180,E1 12846.518,E2 12846.518} C_VEL
LIN {X 0,Y 274.815,Z 737.222,A -85,B 0,C 180,E1 12842.952,E2 12842.952} C_VEL
LIN {X 0,Y 280.516,Z 726.775,A -85,B 0,C 180,E1 12838.884,E2 12838.884} C_VEL
LIN {X 0,Y 287.083,Z 714.684,A -85,B 0,C 180,E1 12835.172,E2 12835.172} C_VEL
LIN {X 0,Y 293.204,Z 703.379,A -85,B 0,C 180,E1 12832.296,E2 12832.296} C_VEL
LIN {X 0,Y 299.213,Z 691.977,A -85,B 0,C 180,E1 12829.844,E2 12829.844} C_VEL
LIN {X 0,Y 305.678,Z 679.197,A -85,B 0,C 180,E1 12827.516,E2 12827.516} C_VEL
LIN {X 0,Y 312.259,Z 665.443,A -85,B 0,C 180,E1 12825.4,E2 12825.4} C_VEL
LIN {X 0,Y 320.327,Z 647.275,A -85,B 0,C 180,E1 12823.087,E2 12823.087} C_VEL
LIN {X 0,Y 327.282,Z 629.644,A -85,B 0,C 180,E1 12821.283,E2 12821.283} C_VEL
LIN {X 0,Y 332.723,Z 614.433,A -85,B 0,C 180,E1 12819.985,E2 12819.985} C_VEL
LIN {X 0,Y 337.711,Z 598.855,A -85,B 0,C 180,E1 12818.869,E2 12818.869} C_VEL
LIN {X 0,Y 342.18,Z 582.969,A -85,B 0,C 180,E1 12817.92,E2 12817.92} C_VEL
LIN {X 0,Y 346.267,Z 566.094,A -85,B 0,C 180,E1 12817.099,E2 12817.099} C_VEL
LIN {X 0,Y 349.765,Z 548.819,A -85,B 0,C 180,E1 12816.434,E2 12816.434} C_VEL
LIN {X 0,Y 352.683,Z 530.329,A -85,B 0,C 180,E1 12815.885,E2 12815.885} C_VEL
LIN {X 0,Y 355.148,Z 505.654,A -85,B 0,C 180,E1 12815.343,E2 12815.343} C_VEL
LIN {X 0,Y 365.762,Z 356.152,A -85,B 0,C 180,E1 12812.631,E2 12812.631} C_VEL
LIN {X 0,Y 358.297,Z 340.185,A -85,B 0,C 180,E1 12810.112,E2 12810.112} C_VEL
LIN {X 0,Y 351.653,Z 327.366,A -85,B 0,C 180,E1 12807.658,E2 12807.658} C_VEL
LIN {X 0,Y 347.377,Z 319.846,A -85,B 0,C 180,E1 12805.946,E2 12805.946} C_VEL
LIN {X 0,Y 340.095,Z 308.94,A -85,B 0,C 180,E1 12802.744,E2 12802.744} C_VEL
LIN {X 0,Y 335.591,Z 302.895,A -85,B 0,C 180,E1 12800.493,E2 12800.493} C_VEL
LIN {X 0,Y 332.382,Z 298.52,A -85,B 0,C 180,E1 12798.686,E2 12798.686} C_VEL
LIN {X 0,Y 328.713,Z 293.564,A -85,B 0,C 180,E1 12796.342,E2 12796.342} C_VEL
LIN {X 0,Y 325.492,Z 289.268,A -85,B 0,C 180,E1 12793.928,E2 12793.928} C_VEL
LIN {X 0,Y 324.589,Z 288.186,A -85,B 0,C 180,E1 12793.177,E2 12793.177} C_VEL
LIN {X 0,Y 321.694,Z 284.735,A -85,B 0,C 180,E1 12790.386,E2 12790.386} C_VEL
LIN {X 0,Y 320.728,Z 282.759,A -85,B 0,C 180,E1 12789.149,E2 12789.149} C_VEL
LIN {X 0,Y 317.033,Z 278.802,A -85,B 0,C 180,E1 12780.723,E2 12780.723} C_VEL
LIN {X 0,Y 317.151,Z 279.15,A -85,B 0,C 180,E1 12777.823,E2 12777.823} C_VEL
LIN {X 0,Y 320.973,Z 283.18,A -85,B 0,C 180,E1 12770.225,E2 12770.225} C_VEL
LIN {X 0,Y 323.254,Z 286.994,A -85,B 0,C 180,E1 12767.677,E2 12767.677} C_VEL
LIN {X 0,Y 325.382,Z 289.066,A -85,B 0,C 180,E1 12765.859,E2 12765.859} C_VEL
LIN {X 0,Y 328.661,Z 293.54,A -85,B 0,C 180,E1 12763.383,E2 12763.383} C_VEL
LIN {X 0,Y 330.168,Z 295.616,A -85,B 0,C 180,E1 12762.372,E2 12762.372} C_VEL
LIN {X 0,Y 333.977,Z 300.614,A -85,B 0,C 180,E1 12760.089,E2 12760.089} C_VEL
LIN {X 0,Y 338.044,Z 306.249,A -85,B 0,C 180,E1 12757.935,E2 12757.935} C_VEL
LIN {X 0,Y 343.472,Z 313.966,A -85,B 0,C 180,E1 12755.399,E2 12755.399} C_VEL
LIN {X 0,Y 351.481,Z 326.072,A -85,B 0,C 180,E1 12752.144,E2 12752.144} C_VEL
LIN {X 0,Y 365.747,Z 347.666,A -85,B 0,C 180,E1 12747.367,E2 12747.367} C_VEL
LIN {X 0,Y 381.003,Z 364.781,A -85,B 0,C 180,E1 12743.388,E2 12743.388} C_VEL
LIN {X 0,Y 402.341,Z 383.247,A -85,B 0,C 180,E1 12738.903,E2 12738.903} C_VEL
LIN {X 0,Y 411.923,Z 391.196,A -85,B 0,C 180,E1 12736.85,E2 12736.85} C_VEL
LIN {X 0,Y 420.903,Z 398.719,A -85,B 0,C 180,E1 12734.789,E2 12734.789} C_VEL
LIN {X 0,Y 430.119,Z 406.715,A -85,B 0,C 180,E1 12732.431,E2 12732.431} C_VEL
LIN {X 0,Y 437.632,Z 413.425,A -85,B 0,C 180,E1 12730.311,E2 12730.311} C_VEL
LIN {X 0,Y 446.468,Z 421.137,A -85,B 0,C 180,E1 12727.704,E2 12727.704} C_VEL
LIN {X 0,Y 455.709,Z 428.984,A -85,B 0,C 180,E1 12724.854,E2 12724.854} C_VEL
LIN {X 0,Y 462.919,Z 434.939,A -85,B 0,C 180,E1 12722.503,E2 12722.503} C_VEL
LIN {X 0,Y 470.055,Z 441.207,A -85,B 0,C 180,E1 12720.03,E2 12720.03} C_VEL
LIN {X 0,Y 475.413,Z 445.416,A -85,B 0,C 180,E1 12718.079,E2 12718.079} C_VEL
LIN {X 0,Y 481.431,Z 450.447,A -85,B 0,C 180,E1 12715.723,E2 12715.723} C_VEL
LIN {X 0,Y 485.976,Z 453.866,A -85,B 0,C 180,E1 12713.844,E2 12713.844} C_VEL
LIN {X 0,Y 491.103,Z 458.321,A -85,B 0,C 180,E1 12711.493,E2 12711.493} C_VEL
LIN {X 0,Y 496.542,Z 462.077,A -85,B 0,C 180,E1 12708.793,E2 12708.793} C_VEL
LIN {X 0,Y 500.593,Z 465.813,A -85,B 0,C 180,E1 12706.475,E2 12706.475} C_VEL
LIN {X 0,Y 504.204,Z 468.412,A -85,B 0,C 180,E1 12704.116,E2 12704.116} C_VEL
LIN {X 0,Y 507.498,Z 470.114,A -85,B 0,C 180,E1 12701.704,E2 12701.704} C_VEL
LIN {X 0,Y 508.661,Z 471.173,A -85,B 0,C 180,E1 12700.62,E2 12700.62} C_VEL
LIN {X 0,Y 510.947,Z 473.58,A -85,B 0,C 180,E1 12698.212,E2 12698.212} C_VEL
LIN {X 0,Y 512.581,Z 475.145,A -85,B 0,C 180,E1 12695.812,E2 12695.812} C_VEL
LIN {X 0,Y 513.83,Z 476.1,A -85,B 0,C 180,E1 12693.235,E2 12693.235} C_VEL
LIN {X 0,Y 514.295,Z 476.405,A -85,B 0,C 180,E1 12690.78,E2 12690.78} C_VEL
LIN {X 0,Y 514.203,Z 476.345,A -85,B 0,C 180,E1 12688.189,E2 12688.189} C_VEL
LIN {X 0,Y 513.349,Z 475.736,A -85,B 0,C 180,E1 12685.644,E2 12685.644} C_VEL
LIN {X 0,Y 511.883,Z 474.54,A -85,B 0,C 180,E1 12683.045,E2 12683.045} C_VEL
LIN {X 0,Y 509.79,Z 472.465,A -85,B 0,C 180,E1 12680.518,E2 12680.518} C_VEL
LIN {X 0,Y 507.643,Z 470.167,A -85,B 0,C 180,E1 12678.412,E2 12678.412} C_VEL
LIN {X 0,Y 504.38,Z 468.514,A -85,B 0,C 180,E1 12676.006,E2 12676.006} C_VEL
LIN {X 0,Y 500.793,Z 465.981,A -85,B 0,C 180,E1 12673.651,E2 12673.651} C_VEL
LIN {X 0,Y 496.657,Z 462.2,A -85,B 0,C 180,E1 12671.273,E2 12671.273} C_VEL
LIN {X 0,Y 493.397,Z 459.913,A -85,B 0,C 180,E1 12669.603,E2 12669.603} C_VEL
LIN {X 0,Y 488.21,Z 455.962,A -85,B 0,C 180,E1 12667.167,E2 12667.167} C_VEL
LIN {X 0,Y 483.536,Z 451.883,A -85,B 0,C 180,E1 12665.118,E2 12665.118} C_VEL
LIN {X 0,Y 477.635,Z 447.43,A -85,B 0,C 180,E1 12662.78,E2 12662.78} C_VEL
LIN {X 0,Y 472.433,Z 442.966,A -85,B 0,C 180,E1 12660.815,E2 12660.815} C_VEL
LIN {X 0,Y 465.973,Z 437.737,A -85,B 0,C 180,E1 12658.535,E2 12658.535} C_VEL
LIN {X 0,Y 460.328,Z 432.97,A -85,B 0,C 180,E1 12656.646,E2 12656.646} C_VEL
LIN {X 0,Y 451.498,Z 425.405,A -85,B 0,C 180,E1 12653.826,E2 12653.826} C_VEL
LIN {X 0,Y 444.007,Z 418.778,A -85,B 0,C 180,E1 12651.548,E2 12651.548} C_VEL
LIN {X 0,Y 436.148,Z 412.028,A -85,B 0,C 180,E1 12649.261,E2 12649.261} C_VEL
LIN {X 0,Y 427.346,Z 404.24,A -85,B 0,C 180,E1 12646.838,E2 12646.838} C_VEL
LIN {X 0,Y 418.408,Z 396.603,A -85,B 0,C 180,E1 12644.635,E2 12644.635} C_VEL
LIN {X 0,Y 410.162,Z 389.743,A -85,B 0,C 180,E1 12642.76,E2 12642.76} C_VEL
LIN {X 0,Y 399.145,Z 380.605,A -85,B 0,C 180,E1 12640.453,E2 12640.453} C_VEL
LIN {X 0,Y 379.125,Z 362.856,A -85,B 0,C 180,E1 12636.165,E2 12636.165} C_VEL
LIN {X 0,Y 364.806,Z 346.424,A -85,B 0,C 180,E1 12632.355,E2 12632.355} C_VEL
LIN {X 0,Y 348.941,Z 322.115,A -85,B 0,C 180,E1 12626.874,E2 12626.874} C_VEL
LIN {X 0,Y 341.284,Z 310.847,A -85,B 0,C 180,E1 12623.619,E2 12623.619} C_VEL
LIN {X 0,Y 336.002,Z 303.378,A -85,B 0,C 180,E1 12621.014,E2 12621.014} C_VEL
LIN {X 0,Y 332.472,Z 298.61,A -85,B 0,C 180,E1 12619.045,E2 12619.045} C_VEL
LIN {X 0,Y 328.766,Z 293.637,A -85,B 0,C 180,E1 12616.687,E2 12616.687} C_VEL
LIN {X 0,Y 325.481,Z 289.254,A -85,B 0,C 180,E1 12614.227,E2 12614.227} C_VEL
LIN {X 0,Y 324.442,Z 288.077,A -85,B 0,C 180,E1 12613.364,E2 12613.364} C_VEL
LIN {X 0,Y 321.588,Z 284.566,A -85,B 0,C 180,E1 12610.57,E2 12610.57} C_VEL
LIN {X 0,Y 320.773,Z 282.786,A -85,B 0,C 180,E1 12609.509,E2 12609.509} C_VEL
LIN {X 0,Y 317.026,Z 278.776,A -85,B 0,C 180,E1 12600.904,E2 12600.904} C_VEL
LIN {X 0,Y 317.199,Z 279.264,A -85,B 0,C 180,E1 12597.832,E2 12597.832} C_VEL
LIN {X 0,Y 320.933,Z 283.089,A -85,B 0,C 180,E1 12590.586,E2 12590.586} C_VEL
LIN {X 0,Y 323.386,Z 287.121,A -85,B 0,C 180,E1 12587.863,E2 12587.863} C_VEL
LIN {X 0,Y 325.323,Z 288.944,A -85,B 0,C 180,E1 12586.22,E2 12586.22} C_VEL
LIN {X 0,Y 328.458,Z 293.325,A -85,B 0,C 180,E1 12583.827,E2 12583.827} C_VEL
LIN {X 0,Y 329.841,Z 295.077,A -85,B 0,C 180,E1 12582.899,E2 12582.899} C_VEL
LIN {X 0,Y 334.027,Z 300.73,A -85,B 0,C 180,E1 12580.366,E2 12580.366} C_VEL
LIN {X 0,Y 337.944,Z 306.09,A -85,B 0,C 180,E1 12578.294,E2 12578.294} C_VEL
LIN {X 0,Y 343.451,Z 313.892,A -85,B 0,C 180,E1 12575.718,E2 12575.718} C_VEL
LIN {X 0,Y 349.074,Z 322.634,A -85,B 0,C 180,E1 12573.366,E2 12573.366} C_VEL
LIN {X 0,Y 355.471,Z 334.573,A -85,B 0,C 180,E1 12570.904,E2 12570.904} C_VEL
LIN {X 0,Y 362.883,Z 349.773,A -85,B 0,C 180,E1 12568.315,E2 12568.315} C_VEL
LIN {X 0,Y 365.834,Z 356.674,A -85,B 0,C 180,E1 12567.333,E2 12567.333} C_VEL
LIN {X 0,Y 364.616,Z 373.344,A -85,B 0,C 180,E1 12567.037,E2 12567.037} C_VEL
LIN {X 0,Y 363.511,Z 381.031,A -85,B 0,C 180,E1 12567.032,E2 12567.032} C_VEL
LIN {X 0,Y 358.613,Z 401.497,A -85,B 0,C 180,E1 12567.499,E2 12567.499} C_VEL
LIN {X 0,Y 357.722,Z 408.095,A -85,B 0,C 180,E1 12567.482,E2 12567.482} C_VEL
LIN {X 0,Y 349.415,Z 518.405,A -85,B 0,C 180,E1 12565.463,E2 12565.463} C_VEL
LIN {X 0,Y 346.824,Z 538.601,A -85,B 0,C 180,E1 12564.957,E2 12564.957} C_VEL
LIN {X 0,Y 342.334,Z 562.204,A -85,B 0,C 180,E1 12564.136,E2 12564.136} C_VEL
LIN {X 0,Y 337.963,Z 580.307,A -85,B 0,C 180,E1 12563.289,E2 12563.289} C_VEL
LIN {X 0,Y 333.366,Z 596.556,A -85,B 0,C 180,E1 12562.347,E2 12562.347} C_VEL
LIN {X 0,Y 328.231,Z 612.417,A -85,B 0,C 180,E1 12561.237,E2 12561.237} C_VEL
LIN {X 0,Y 322.617,Z 627.856,A -85,B 0,C 180,E1 12559.945,E2 12559.945} C_VEL
LIN {X 0,Y 316.6,Z 642.834,A -85,B 0,C 180,E1 12558.451,E2 12558.451} C_VEL
LIN {X 0,Y 309.682,Z 658.563,A -85,B 0,C 180,E1 12556.583,E2 12556.583} C_VEL
LIN {X 0,Y 300.77,Z 677.022,A -85,B 0,C 180,E1 12553.872,E2 12553.872} C_VEL
LIN {X 0,Y 293.999,Z 690.02,A -85,B 0,C 180,E1 12551.537,E2 12551.537} C_VEL
LIN {X 0,Y 287.514,Z 701.906,A -85,B 0,C 180,E1 12549.004,E2 12549.004} C_VEL
LIN {X 0,Y 281.603,Z 712.401,A -85,B 0,C 180,E1 12546.362,E2 12546.362} C_VEL
LIN {X 0,Y 275.938,Z 722.291,A -85,B 0,C 180,E1 12543.416,E2 12543.416} C_VEL
LIN {X 0,Y 270.684,Z 731.475,A -85,B 0,C 180,E1 12540.153,E2 12540.153} C_VEL
LIN {X 0,Y 265.531,Z 740.795,A -85,B 0,C 180,E1 12536.137,E2 12536.137} C_VEL
LIN {X 0,Y 261.04,Z 749.447,A -85,B 0,C 180,E1 12531.336,E2 12531.336} C_VEL
LIN {X 0,Y 258.503,Z 755.067,A -85,B 0,C 180,E1 12527.325,E2 12527.325} C_VEL
LIN {X 0,Y 256.957,Z 759.345,A -85,B 0,C 180,E1 12523.388,E2 12523.388} C_VEL
LIN {X 0,Y 256.202,Z 762.352,A -85,B 0,C 180,E1 12519.66,E2 12519.66} C_VEL
LIN {X 0,Y 255.966,Z 764.334,A -85,B 0,C 180,E1 12516.053,E2 12516.053} C_VEL
LIN {X 0,Y 255.965,Z 765.412,A -85,B 0,C 180,E1 12512.462,E2 12512.462} C_VEL
LIN {X 0,Y 255.983,Z 765.591,A -85,B 0,C 180,E1 12508.881,E2 12508.881} C_VEL
LIN {X 0,Y 255.944,Z 764.756,A -85,B 0,C 180,E1 12505.009,E2 12505.009} C_VEL
LIN {X 0,Y 256.136,Z 762.779,A -85,B 0,C 180,E1 12500.987,E2 12500.987} C_VEL
LIN {X 0,Y 256.806,Z 759.871,A -85,B 0,C 180,E1 12497.179,E2 12497.179} C_VEL
LIN {X 0,Y 258.178,Z 755.879,A -85,B 0,C 180,E1 12493.348,E2 12493.348} C_VEL
LIN {X 0,Y 260.392,Z 750.778,A -85,B 0,C 180,E1 12489.546,E2 12489.546} C_VEL
LIN {X 0,Y 263.5,Z 744.531,A -85,B 0,C 180,E1 12485.81,E2 12485.81} C_VEL
LIN {X 0,Y 267.555,Z 737.043,A -85,B 0,C 180,E1 12482.155,E2 12482.155} C_VEL
LIN {X 0,Y 273.549,Z 726.593,A -85,B 0,C 180,E1 12477.997,E2 12477.997} C_VEL
LIN {X 0,Y 280.413,Z 714.505,A -85,B 0,C 180,E1 12474.218,E2 12474.218} C_VEL
LIN {X 0,Y 286.632,Z 703.489,A -85,B 0,C 180,E1 12471.366,E2 12471.366} C_VEL
LIN {X 0,Y 293.035,Z 691.799,A -85,B 0,C 180,E1 12468.817,E2 12468.817} C_VEL
LIN {X 0,Y 299.473,Z 679.519,A -85,B 0,C 180,E1 12466.551,E2 12466.551} C_VEL
LIN {X 0,Y 306.088,Z 666.172,A -85,B 0,C 180,E1 12464.466,E2 12464.466} C_VEL
LIN {X 0,Y 313.683,Z 649.742,A -85,B 0,C 180,E1 12462.318,E2 12462.318} C_VEL
LIN {X 0,Y 321.688,Z 630.314,A -85,B 0,C 180,E1 12460.28,E2 12460.28} C_VEL
LIN {X 0,Y 327.598,Z 614.256,A -85,B 0,C 180,E1 12458.904,E2 12458.904} C_VEL
LIN {X 0,Y 332.716,Z 598.679,A -85,B 0,C 180,E1 12457.789,E2 12457.789} C_VEL
LIN {X 0,Y 337.296,Z 582.793,A -85,B 0,C 180,E1 12456.843,E2 12456.843} C_VEL
LIN {X 0,Y 341.482,Z 565.918,A -85,B 0,C 180,E1 12456.024,E2 12456.024} C_VEL
LIN {X 0,Y 345.082,Z 548.529,A -85,B 0,C 180,E1 12455.358,E2 12455.358} C_VEL
LIN {X 0,Y 348.087,Z 529.859,A -85,B 0,C 180,E1 12454.808,E2 12454.808} C_VEL
LIN {X 0,Y 350.69,Z 503.823,A -85,B 0,C 180,E1 12454.244,E2 12454.244} C_VEL
LIN {X 0,Y 361.247,Z 359.755,A -85,B 0,C 180,E1 12451.636,E2 12451.636} C_VEL
LIN {X 0,Y 354.224,Z 344.497,A -85,B 0,C 180,E1 12449.139,E2 12449.139} C_VEL
LIN {X 0,Y 347.831,Z 331.91,A -85,B 0,C 180,E1 12446.644,E2 12446.644} C_VEL
LIN {X 0,Y 343.788,Z 324.944,A -85,B 0,C 180,E1 12444.944,E2 12444.944} C_VEL
LIN {X 0,Y 337.191,Z 315.153,A -85,B 0,C 180,E1 12441.894,E2 12441.894} C_VEL
LIN {X 0,Y 333.546,Z 310.063,A -85,B 0,C 180,E1 12439.983,E2 12439.983} C_VEL
LIN {X 0,Y 330.564,Z 305.905,A -85,B 0,C 180,E1 12438.244,E2 12438.244} C_VEL
LIN {X 0,Y 327.118,Z 301.132,A -85,B 0,C 180,E1 12435.968,E2 12435.968} C_VEL
LIN {X 0,Y 323.923,Z 296.684,A -85,B 0,C 180,E1 12433.477,E2 12433.477} C_VEL
LIN {X 0,Y 320.334,Z 292.284,A -85,B 0,C 180,E1 12429.976,E2 12429.976} C_VEL
LIN {X 0,Y 319.463,Z 290.565,A -85,B 0,C 180,E1 12428.822,E2 12428.822} C_VEL
LIN {X 0,Y 316.046,Z 286.726,A -85,B 0,C 180,E1 12420.544,E2 12420.544} C_VEL
LIN {X 0,Y 316.2,Z 287.186,A -85,B 0,C 180,E1 12417.644,E2 12417.644} C_VEL
LIN {X 0,Y 319.711,Z 290.889,A -85,B 0,C 180,E1 12410.55,E2 12410.55} C_VEL
LIN {X 0,Y 322.097,Z 294.892,A -85,B 0,C 180,E1 12407.814,E2 12407.814} C_VEL
LIN {X 0,Y 323.982,Z 296.806,A -85,B 0,C 180,E1 12406.162,E2 12406.162} C_VEL
LIN {X 0,Y 327.445,Z 301.47,A -85,B 0,C 180,E1 12403.502,E2 12403.502} C_VEL
LIN {X 0,Y 332.332,Z 308.313,A -85,B 0,C 180,E1 12400.399,E2 12400.399} C_VEL
LIN {X 0,Y 336.251,Z 313.856,A -85,B 0,C 180,E1 12398.271,E2 12398.271} C_VEL
LIN {X 0,Y 341.321,Z 321.277,A -85,B 0,C 180,E1 12395.833,E2 12395.833} C_VEL
LIN {X 0,Y 349.074,Z 333.247,A -85,B 0,C 180,E1 12392.588,E2 12392.588} C_VEL
LIN {X 0,Y 362.55,Z 354.088,A -85,B 0,C 180,E1 12387.933,E2 12387.933} C_VEL
LIN {X 0,Y 377.425,Z 371.119,A -85,B 0,C 180,E1 12383.928,E2 12383.928} C_VEL
LIN {X 0,Y 399.496,Z 390.404,A -85,B 0,C 180,E1 12379.213,E2 12379.213} C_VEL
LIN {X 0,Y 409.871,Z 398.905,A -85,B 0,C 180,E1 12377.021,E2 12377.021} C_VEL
LIN {X 0,Y 416.859,Z 404.724,A -85,B 0,C 180,E1 12375.435,E2 12375.435} C_VEL
LIN {X 0,Y 425.864,Z 412.324,A -85,B 0,C 180,E1 12373.244,E2 12373.244} C_VEL
LIN {X 0,Y 434.702,Z 420.094,A -85,B 0,C 180,E1 12370.821,E2 12370.821} C_VEL
LIN {X 0,Y 444.28,Z 428.426,A -85,B 0,C 180,E1 12368.028,E2 12368.028} C_VEL
LIN {X 0,Y 453.465,Z 436.17,A -85,B 0,C 180,E1 12365.219,E2 12365.219} C_VEL
LIN {X 0,Y 460.836,Z 442.287,A -85,B 0,C 180,E1 12362.844,E2 12362.844} C_VEL
LIN {X 0,Y 468.405,Z 448.836,A -85,B 0,C 180,E1 12360.246,E2 12360.246} C_VEL
LIN {X 0,Y 473.885,Z 453.146,A -85,B 0,C 180,E1 12358.252,E2 12358.252} C_VEL
LIN {X 0,Y 480.039,Z 458.235,A -85,B 0,C 180,E1 12355.864,E2 12355.864} C_VEL
LIN {X 0,Y 484.444,Z 461.517,A -85,B 0,C 180,E1 12354.053,E2 12354.053} C_VEL
LIN {X 0,Y 489.67,Z 466.034,A -85,B 0,C 180,E1 12351.688,E2 12351.688} C_VEL
LIN {X 0,Y 494.754,Z 469.305,A -85,B 0,C 180,E1 12349.231,E2 12349.231} C_VEL
LIN {X 0,Y 498.854,Z 473.233,A -85,B 0,C 180,E1 12346.894,E2 12346.894} C_VEL
LIN {X 0,Y 502.825,Z 476.136,A -85,B 0,C 180,E1 12344.391,E2 12344.391} C_VEL
LIN {X 0,Y 506.143,Z 477.92,A -85,B 0,C 180,E1 12341.97,E2 12341.97} C_VEL
LIN {X 0,Y 507.369,Z 478.806,A -85,B 0,C 180,E1 12340.904,E2 12340.904} C_VEL
LIN {X 0,Y 509.661,Z 481.231,A -85,B 0,C 180,E1 12338.574,E2 12338.574} C_VEL
LIN {X 0,Y 511.455,Z 482.974,A -85,B 0,C 180,E1 12336.059,E2 12336.059} C_VEL
LIN {X 0,Y 512.737,Z 483.956,A -85,B 0,C 180,E1 12333.577,E2 12333.577} C_VEL
LIN {X 0,Y 513.299,Z 484.342,A -85,B 0,C 180,E1 12331.004,E2 12331.004} C_VEL
LIN {X 0,Y 513.285,Z 484.33,A -85,B 0,C 180,E1 12328.549,E2 12328.549} C_VEL
LIN {X 0,Y 512.513,Z 483.805,A -85,B 0,C 180,E1 12325.973,E2 12325.973} C_VEL
LIN {X 0,Y 511.211,Z 482.748,A -85,B 0,C 180,E1 12323.487,E2 12323.487} C_VEL
LIN {X 0,Y 509.206,Z 480.839,A -85,B 0,C 180,E1 12320.963,E2 12320.963} C_VEL
LIN {X 0,Y 507.133,Z 478.486,A -85,B 0,C 180,E1 12318.861,E2 12318.861} C_VEL
LIN {X 0,Y 503.594,Z 476.593,A -85,B 0,C 180,E1 12316.148,E2 12316.148} C_VEL
LIN {X 0,Y 499.938,Z 474.096,A -85,B 0,C 180,E1 12313.742,E2 12313.742} C_VEL
LIN {X 0,Y 495.68,Z 470.309,A -85,B 0,C 180,E1 12311.295,E2 12311.295} C_VEL
LIN {X 0,Y 493.381,Z 468.519,A -85,B 0,C 180,E1 12310.097,E2 12310.097} C_VEL
LIN {X 0,Y 488.428,Z 465.046,A -85,B 0,C 180,E1 12307.717,E2 12307.717} C_VEL
LIN {X 0,Y 482.167,Z 459.676,A -85,B 0,C 180,E1 12304.977,E2 12304.977} C_VEL
LIN {X 0,Y 476.196,Z 455.203,A -85,B 0,C 180,E1 12302.627,E2 12302.627} C_VEL
LIN {X 0,Y 470.843,Z 450.657,A -85,B 0,C 180,E1 12300.627,E2 12300.627} C_VEL
LIN {X 0,Y 464.196,Z 445.295,A -85,B 0,C 180,E1 12298.297,E2 12298.297} C_VEL
LIN {X 0,Y 458.362,Z 440.404,A -85,B 0,C 180,E1 12296.357,E2 12296.357} C_VEL
LIN {X 0,Y 449.467,Z 432.841,A -85,B 0,C 180,E1 12293.544,E2 12293.544} C_VEL
LIN {X 0,Y 440.432,Z 425.025,A -85,B 0,C 180,E1 12290.832,E2 12290.832} C_VEL
LIN {X 0,Y 432.648,Z 418.1,A -85,B 0,C 180,E1 12288.586,E2 12288.586} C_VEL
LIN {X 0,Y 424.728,Z 411.326,A -85,B 0,C 180,E1 12286.477,E2 12286.477} C_VEL
LIN {X 0,Y 416.444,Z 404.365,A -85,B 0,C 180,E1 12284.467,E2 12284.467} C_VEL
LIN {X 0,Y 409.087,Z 398.274,A -85,B 0,C 180,E1 12282.804,E2 12282.804} C_VEL
LIN {X 0,Y 397.874,Z 389.104,A -85,B 0,C 180,E1 12280.467,E2 12280.467} C_VEL
LIN {X 0,Y 376.497,Z 370.155,A -85,B 0,C 180,E1 12275.845,E2 12275.845} C_VEL
LIN {X 0,Y 362.087,Z 353.468,A -85,B 0,C 180,E1 12271.926,E2 12271.926} C_VEL
LIN {X 0,Y 346.308,Z 328.86,A -85,B 0,C 180,E1 12266.308,E2 12266.308} C_VEL
LIN {X 0,Y 338.686,Z 317.346,A -85,B 0,C 180,E1 12262.936,E2 12262.936} C_VEL
LIN {X 0,Y 333.794,Z 310.364,A -85,B 0,C 180,E1 12260.425,E2 12260.425} C_VEL
LIN {X 0,Y 330.513,Z 305.842,A -85,B 0,C 180,E1 12258.521,E2 12258.521} C_VEL
LIN {X 0,Y 327.07,Z 301.104,A -85,B 0,C 180,E1 12256.244,E2 12256.244} C_VEL
LIN {X 0,Y 323.792,Z 296.428,A -85,B 0,C 180,E1 12253.665,E2 12253.665} C_VEL
LIN {X 0,Y 320.519,Z 292.677,A -85,B 0,C 180,E1 12250.515,E2 12250.515} C_VEL
LIN {X 0,Y 319.506,Z 290.605,A -85,B 0,C 180,E1 12249.184,E2 12249.184} C_VEL
LIN {X 0,Y 316.05,Z 286.727,A -85,B 0,C 180,E1 12240.906,E2 12240.906} C_VEL
LIN {X 0,Y 316.222,Z 287.229,A -85,B 0,C 180,E1 12237.825,E2 12237.825} C_VEL
LIN {X 0,Y 319.735,Z 290.947,A -85,B 0,C 180,E1 12230.823,E2 12230.823} C_VEL
LIN {X 0,Y 322.227,Z 295.017,A -85,B 0,C 180,E1 12228,E2 12228} C_VEL
LIN {X 0,Y 323.923,Z 296.686,A -85,B 0,C 180,E1 12226.523,E2 12226.523} C_VEL
LIN {X 0,Y 327.118,Z 301.136,A -85,B 0,C 180,E1 12224.032,E2 12224.032} C_VEL
LIN {X 0,Y 332.169,Z 308.095,A -85,B 0,C 180,E1 12220.8,E2 12220.8} C_VEL
LIN {X 0,Y 336.23,Z 313.813,A -85,B 0,C 180,E1 12218.59,E2 12218.59} C_VEL
LIN {X 0,Y 341.384,Z 321.344,A -85,B 0,C 180,E1 12216.113,E2 12216.113} C_VEL
LIN {X 0,Y 346.436,Z 329.375,A -85,B 0,C 180,E1 12213.932,E2 12213.932} C_VEL
LIN {X 0,Y 352.483,Z 340.98,A -85,B 0,C 180,E1 12211.515,E2 12211.515} C_VEL
LIN {X 0,Y 359.508,Z 355.788,A -85,B 0,C 180,E1 12208.964,E2 12208.964} C_VEL
LIN {X 0,Y 361.283,Z 360.261,A -85,B 0,C 180,E1 12208.336,E2 12208.336} C_VEL
LIN {X 0,Y 357.722,Z 408.095,A -85,B 0,C 180,E1 12207.482,E2 12207.482} C_VEL
LIN {X 0,Y 356.615,Z 415.782,A -85,B 0,C 180,E1 12207.478,E2 12207.478} C_VEL
LIN {X 0,Y 351.717,Z 436.239,A -85,B 0,C 180,E1 12207.967,E2 12207.967} C_VEL
LIN {X 0,Y 350.818,Z 442.837,A -85,B 0,C 180,E1 12207.952,E2 12207.952} C_VEL
LIN {X 0,Y 344.892,Z 518.631,A -85,B 0,C 180,E1 12206.552,E2 12206.552} C_VEL
LIN {X 0,Y 342.028,Z 540.151,A -85,B 0,C 180,E1 12206.009,E2 12206.009} C_VEL
LIN {X 0,Y 337.518,Z 562.772,A -85,B 0,C 180,E1 12205.209,E2 12205.209} C_VEL
LIN {X 0,Y 333.219,Z 580.131,A -85,B 0,C 180,E1 12204.398,E2 12204.398} C_VEL
LIN {X 0,Y 328.509,Z 596.38,A -85,B 0,C 180,E1 12203.459,E2 12203.459} C_VEL
LIN {X 0,Y 323.243,Z 612.24,A -85,B 0,C 180,E1 12202.352,E2 12202.352} C_VEL
LIN {X 0,Y 317.476,Z 627.68,A -85,B 0,C 180,E1 12201.061,E2 12201.061} C_VEL
LIN {X 0,Y 311.288,Z 642.657,A -85,B 0,C 180,E1 12199.567,E2 12199.567} C_VEL
LIN {X 0,Y 303.877,Z 659.015,A -85,B 0,C 180,E1 12197.612,E2 12197.612} C_VEL
LIN {X 0,Y 294.962,Z 676.845,A -85,B 0,C 180,E1 12194.967,E2 12194.967} C_VEL
LIN {X 0,Y 287.834,Z 690.054,A -85,B 0,C 180,E1 12192.569,E2 12192.569} C_VEL
LIN {X 0,Y 281.222,Z 701.728,A -85,B 0,C 180,E1 12190.05,E2 12190.05} C_VEL
LIN {X 0,Y 275.069,Z 712.222,A -85,B 0,C 180,E1 12187.371,E2 12187.371} C_VEL
LIN {X 0,Y 269.151,Z 722.113,A -85,B 0,C 180,E1 12184.374,E2 12184.374} C_VEL
LIN {X 0,Y 263.642,Z 731.296,A -85,B 0,C 180,E1 12181.046,E2 12181.046} C_VEL
LIN {X 0,Y 258.215,Z 740.616,A -85,B 0,C 180,E1 12176.936,E2 12176.936} C_VEL
LIN {X 0,Y 253.45,Z 749.269,A -85,B 0,C 180,E1 12172.008,E2 12172.008} C_VEL
LIN {X 0,Y 250.739,Z 754.889,A -85,B 0,C 180,E1 12167.879,E2 12167.879} C_VEL
LIN {X 0,Y 249.101,Z 759.065,A -85,B 0,C 180,E1 12163.934,E2 12163.934} C_VEL
LIN {X 0,Y 248.239,Z 762.176,A -85,B 0,C 180,E1 12159.973,E2 12159.973} C_VEL
LIN {X 0,Y 247.972,Z 764.159,A -85,B 0,C 180,E1 12156.249,E2 12156.249} C_VEL
LIN {X 0,Y 247.965,Z 765.237,A -85,B 0,C 180,E1 12152.542,E2 12152.542} C_VEL
LIN {X 0,Y 247.984,Z 765.416,A -85,B 0,C 180,E1 12148.845,E2 12148.845} C_VEL
LIN {X 0,Y 247.946,Z 764.605,A -85,B 0,C 180,E1 12144.911,E2 12144.911} C_VEL
LIN {X 0,Y 248.16,Z 762.623,A -85,B 0,C 180,E1 12140.727,E2 12140.727} C_VEL
LIN {X 0,Y 248.901,Z 759.693,A -85,B 0,C 180,E1 12136.765,E2 12136.765} C_VEL
LIN {X 0,Y 250.389,Z 755.702,A -85,B 0,C 180,E1 12132.814,E2 12132.814} C_VEL
LIN {X 0,Y 252.759,Z 750.607,A -85,B 0,C 180,E1 12128.904,E2 12128.904} C_VEL
LIN {X 0,Y 256.065,Z 744.352,A -85,B 0,C 180,E1 12125.06,E2 12125.06} C_VEL
LIN {X 0,Y 260.35,Z 736.864,A -85,B 0,C 180,E1 12121.314,E2 12121.314} C_VEL
LIN {X 0,Y 266.647,Z 726.417,A -85,B 0,C 180,E1 12117.067,E2 12117.067} C_VEL
LIN {X 0,Y 273.827,Z 714.327,A -85,B 0,C 180,E1 12113.218,E2 12113.218} C_VEL
LIN {X 0,Y 280.306,Z 703.311,A -85,B 0,C 180,E1 12110.325,E2 12110.325} C_VEL
LIN {X 0,Y 286.955,Z 691.621,A -85,B 0,C 180,E1 12107.746,E2 12107.746} C_VEL
LIN {X 0,Y 293.89,Z 678.842,A -85,B 0,C 180,E1 12105.375,E2 12105.375} C_VEL
LIN {X 0,Y 300.74,Z 665.434,A -85,B 0,C 180,E1 12103.279,E2 12103.279} C_VEL
LIN {X 0,Y 309.192,Z 647.63,A -85,B 0,C 180,E1 12100.974,E2 12100.974} C_VEL
LIN {X 0,Y 316.85,Z 629.291,A -85,B 0,C 180,E1 12099.086,E2 12099.086} C_VEL
LIN {X 0,Y 322.594,Z 614.08,A -85,B 0,C 180,E1 12097.789,E2 12097.789} C_VEL
LIN {X 0,Y 327.843,Z 598.503,A -85,B 0,C 180,E1 12096.677,E2 12096.677} C_VEL
LIN {X 0,Y 332.537,Z 582.617,A -85,B 0,C 180,E1 12095.734,E2 12095.734} C_VEL
LIN {X 0,Y 336.82,Z 565.743,A -85,B 0,C 180,E1 12094.918,E2 12094.918} C_VEL
LIN {X 0,Y 340.501,Z 548.354,A -85,B 0,C 180,E1 12094.257,E2 12094.257} C_VEL
LIN {X 0,Y 343.572,Z 529.684,A -85,B 0,C 180,E1 12093.709,E2 12093.709} C_VEL
LIN {X 0,Y 346.241,Z 503.648,A -85,B 0,C 180,E1 12093.147,E2 12093.147} C_VEL
LIN {X 0,Y 356.842,Z 363.38,A -85,B 0,C 180,E1 12090.616,E2 12090.616} C_VEL
LIN {X 0,Y 350.449,Z 349.314,A -85,B 0,C 180,E1 12088.224,E2 12088.224} C_VEL
LIN {X 0,Y 344.825,Z 337.981,A -85,B 0,C 180,E1 12085.921,E2 12085.921} C_VEL
LIN {X 0,Y 341.143,Z 331.556,A -85,B 0,C 180,E1 12084.309,E2 12084.309} C_VEL
LIN {X 0,Y 334.997,Z 322.192,A -85,B 0,C 180,E1 12081.355,E2 12081.355} C_VEL
LIN {X 0,Y 331.384,Z 317.03,A -85,B 0,C 180,E1 12079.385,E2 12079.385} C_VEL
LIN {X 0,Y 328.766,Z 313.288,A -85,B 0,C 180,E1 12077.798,E2 12077.798} C_VEL
LIN {X 0,Y 325.538,Z 308.698,A -85,B 0,C 180,E1 12075.59,E2 12075.59} C_VEL
LIN {X 0,Y 322.042,Z 303.79,A -85,B 0,C 180,E1 12072.735,E2 12072.735} C_VEL
LIN {X 0,Y 319.126,Z 300.114,A -85,B 0,C 180,E1 12069.741,E2 12069.741} C_VEL
LIN {X 0,Y 318.21,Z 298.37,A -85,B 0,C 180,E1 12068.493,E2 12068.493} C_VEL
LIN {X 0,Y 315.071,Z 294.669,A -85,B 0,C 180,E1 12060.546,E2 12060.546} C_VEL
LIN {X 0,Y 315.195,Z 295.073,A -85,B 0,C 180,E1 12057.818,E2 12057.818} C_VEL
LIN {X 0,Y 318.519,Z 298.752,A -85,B 0,C 180,E1 12050.787,E2 12050.787} C_VEL
LIN {X 0,Y 320.941,Z 302.789,A -85,B 0,C 180,E1 12047.952,E2 12047.952} C_VEL
LIN {X 0,Y 322.591,Z 304.54,A -85,B 0,C 180,E1 12046.466,E2 12046.466} C_VEL
LIN {X 0,Y 326.685,Z 310.34,A -85,B 0,C 180,E1 12043.279,E2 12043.279} C_VEL
LIN {X 0,Y 330.56,Z 315.787,A -85,B 0,C 180,E1 12040.795,E2 12040.795} C_VEL
LIN {X 0,Y 334.549,Z 321.568,A -85,B 0,C 180,E1 12038.569,E2 12038.569} C_VEL
LIN {X 0,Y 339.871,Z 329.683,A -85,B 0,C 180,E1 12035.954,E2 12035.954} C_VEL
LIN {X 0,Y 346.609,Z 340.33,A -85,B 0,C 180,E1 12033.069,E2 12033.069} C_VEL
LIN {X 0,Y 359.617,Z 360.817,A -85,B 0,C 180,E1 12028.438,E2 12028.438} C_VEL
LIN {X 0,Y 374.406,Z 377.999,A -85,B 0,C 180,E1 12024.348,E2 12024.348} C_VEL
LIN {X 0,Y 396.608,Z 397.553,A -85,B 0,C 180,E1 12019.52,E2 12019.52} C_VEL
LIN {X 0,Y 407.611,Z 406.437,A -85,B 0,C 180,E1 12017.244,E2 12017.244} C_VEL
LIN {X 0,Y 416.569,Z 413.865,A -85,B 0,C 180,E1 12015.212,E2 12015.212} C_VEL
LIN {X 0,Y 425.333,Z 421.237,A -85,B 0,C 180,E1 12013.07,E2 12013.07} C_VEL
LIN {X 0,Y 433.043,Z 427.937,A -85,B 0,C 180,E1 12010.97,E2 12010.97} C_VEL
LIN {X 0,Y 442.769,Z 436.343,A -85,B 0,C 180,E1 12008.146,E2 12008.146} C_VEL
LIN {X 0,Y 452.089,Z 444.168,A -85,B 0,C 180,E1 12005.301,E2 12005.301} C_VEL
LIN {X 0,Y 459.381,Z 450.12,A -85,B 0,C 180,E1 12002.962,E2 12002.962} C_VEL
LIN {X 0,Y 466.557,Z 456.347,A -85,B 0,C 180,E1 12000.51,E2 12000.51} C_VEL
LIN {X 0,Y 472.316,Z 460.835,A -85,B 0,C 180,E1 11998.441,E2 11998.441} C_VEL
LIN {X 0,Y 478.554,Z 465.953,A -85,B 0,C 180,E1 11996.046,E2 11996.046} C_VEL
LIN {X 0,Y 483.075,Z 469.327,A -85,B 0,C 180,E1 11994.191,E2 11994.191} C_VEL
LIN {X 0,Y 488.393,Z 473.862,A -85,B 0,C 180,E1 11991.81,E2 11991.81} C_VEL
LIN {X 0,Y 493.659,Z 477.307,A -85,B 0,C 180,E1 11989.275,E2 11989.275} C_VEL
LIN {X 0,Y 497.781,Z 481.187,A -85,B 0,C 180,E1 11986.931,E2 11986.931} C_VEL
LIN {X 0,Y 501.79,Z 484.072,A -85,B 0,C 180,E1 11984.421,E2 11984.421} C_VEL
LIN {X 0,Y 505.121,Z 485.852,A -85,B 0,C 180,E1 11981.995,E2 11981.995} C_VEL
LIN {X 0,Y 506.353,Z 486.786,A -85,B 0,C 180,E1 11980.926,E2 11980.926} C_VEL
LIN {X 0,Y 508.658,Z 489.184,A -85,B 0,C 180,E1 11978.591,E2 11978.591} C_VEL
LIN {X 0,Y 510.469,Z 490.917,A -85,B 0,C 180,E1 11976.071,E2 11976.071} C_VEL
LIN {X 0,Y 511.755,Z 491.896,A -85,B 0,C 180,E1 11973.584,E2 11973.584} C_VEL
LIN {X 0,Y 512.323,Z 492.282,A -85,B 0,C 180,E1 11971.006,E2 11971.006} C_VEL
LIN {X 0,Y 512.309,Z 492.271,A -85,B 0,C 180,E1 11968.546,E2 11968.546} C_VEL
LIN {X 0,Y 511.532,Z 491.746,A -85,B 0,C 180,E1 11965.965,E2 11965.965} C_VEL
LIN {X 0,Y 510.225,Z 490.692,A -85,B 0,C 180,E1 11963.474,E2 11963.474} C_VEL
LIN {X 0,Y 508.203,Z 488.789,A -85,B 0,C 180,E1 11960.945,E2 11960.945} C_VEL
LIN {X 0,Y 506.117,Z 486.472,A -85,B 0,C 180,E1 11958.838,E2 11958.838} C_VEL
LIN {X 0,Y 502.585,Z 484.544,A -85,B 0,C 180,E1 11956.138,E2 11956.138} C_VEL
LIN {X 0,Y 498.881,Z 482.046,A -85,B 0,C 180,E1 11953.706,E2 11953.706} C_VEL
LIN {X 0,Y 494.587,Z 478.292,A -85,B 0,C 180,E1 11951.252,E2 11951.252} C_VEL
LIN {X 0,Y 492.273,Z 476.442,A -85,B 0,C 180,E1 11950.051,E2 11950.051} C_VEL
LIN {X 0,Y 487.188,Z 472.927,A -85,B 0,C 180,E1 11947.625,E2 11947.625} C_VEL
LIN {X 0,Y 481.124,Z 467.685,A -85,B 0,C 180,E1 11944.974,E2 11944.974} C_VEL
LIN {X 0,Y 475.15,Z 463.312,A -85,B 0,C 180,E1 11942.629,E2 11942.629} C_VEL
LIN {X 0,Y 469.361,Z 458.425,A -85,B 0,C 180,E1 11940.48,E2 11940.48} C_VEL
LIN {X 0,Y 462.645,Z 453.071,A -85,B 0,C 180,E1 11938.144,E2 11938.144} C_VEL
LIN {X 0,Y 456.958,Z 448.291,A -85,B 0,C 180,E1 11936.253,E2 11936.253} C_VEL
LIN {X 0,Y 448.288,Z 440.937,A -85,B 0,C 180,E1 11933.522,E2 11933.522} C_VEL
LIN {X 0,Y 440.54,Z 434.277,A -85,B 0,C 180,E1 11931.191,E2 11931.191} C_VEL
LIN {X 0,Y 431.89,Z 426.857,A -85,B 0,C 180,E1 11928.701,E2 11928.701} C_VEL
LIN {X 0,Y 423.308,Z 419.514,A -85,B 0,C 180,E1 11926.428,E2 11926.428} C_VEL
LIN {X 0,Y 415.264,Z 412.785,A -85,B 0,C 180,E1 11924.482,E2 11924.482} C_VEL
LIN {X 0,Y 405.532,Z 404.781,A -85,B 0,C 180,E1 11922.308,E2 11922.308} C_VEL
LIN {X 0,Y 394.818,Z 396.107,A -85,B 0,C 180,E1 11920.121,E2 11920.121} C_VEL
LIN {X 0,Y 373.489,Z 377.034,A -85,B 0,C 180,E1 11915.423,E2 11915.423} C_VEL
LIN {X 0,Y 359.162,Z 360.197,A -85,B 0,C 180,E1 11911.419,E2 11911.419} C_VEL
LIN {X 0,Y 343.803,Z 335.74,A -85,B 0,C 180,E1 11905.772,E2 11905.772} C_VEL
LIN {X 0,Y 335.825,Z 323.289,A -85,B 0,C 180,E1 11902.08,E2 11902.08} C_VEL
LIN {X 0,Y 330.839,Z 316.213,A -85,B 0,C 180,E1 11899.372,E2 11899.372} C_VEL
LIN {X 0,Y 328.584,Z 313.062,A -85,B 0,C 180,E1 11897.991,E2 11897.991} C_VEL
LIN {X 0,Y 325.492,Z 308.667,A -85,B 0,C 180,E1 11895.867,E2 11895.867} C_VEL
LIN {X 0,Y 322.105,Z 303.844,A -85,B 0,C 180,E1 11893.098,E2 11893.098} C_VEL
LIN {X 0,Y 319.166,Z 300.23,A -85,B 0,C 180,E1 11890.104,E2 11890.104} C_VEL
LIN {X 0,Y 318.251,Z 298.417,A -85,B 0,C 180,E1 11888.856,E2 11888.856} C_VEL
LIN {X 0,Y 315.067,Z 294.633,A -85,B 0,C 180,E1 11880.727,E2 11880.727} C_VEL
LIN {X 0,Y 315.275,Z 295.288,A -85,B 0,C 180,E1 11877.637,E2 11877.637} C_VEL
LIN {X 0,Y 318.543,Z 298.798,A -85,B 0,C 180,E1 11871.061,E2 11871.061} C_VEL
LIN {X 0,Y 321.069,Z 302.911,A -85,B 0,C 180,E1 11868.139,E2 11868.139} C_VEL
LIN {X 0,Y 322.626,Z 304.605,A -85,B 0,C 180,E1 11866.742,E2 11866.742} C_VEL
LIN {X 0,Y 326.61,Z 310.208,A -85,B 0,C 180,E1 11863.641,E2 11863.641} C_VEL
LIN {X 0,Y 330.537,Z 315.783,A -85,B 0,C 180,E1 11861.114,E2 11861.114} C_VEL
LIN {X 0,Y 334.448,Z 321.413,A -85,B 0,C 180,E1 11858.93,E2 11858.93} C_VEL
LIN {X 0,Y 339.59,Z 329.199,A -85,B 0,C 180,E1 11856.394,E2 11856.394} C_VEL
LIN {X 0,Y 343.922,Z 336.288,A -85,B 0,C 180,E1 11854.468,E2 11854.468} C_VEL
LIN {X 0,Y 349.584,Z 347.487,A -85,B 0,C 180,E1 11852.118,E2 11852.118} C_VEL
LIN {X 0,Y 356.181,Z 361.802,A -85,B 0,C 180,E1 11849.625,E2 11849.625} C_VEL
LIN {X 0,Y 356.851,Z 363.796,A -85,B 0,C 180,E1 11849.366,E2 11849.366} C_VEL
LIN {X 0,Y 350.818,Z 442.837,A -85,B 0,C 180,E1 11847.952,E2 11847.952} C_VEL
LIN {X 0,Y 349.703,Z 450.524,A -85,B 0,C 180,E1 11847.952,E2 11847.952} C_VEL
LIN {X 0,Y 344.814,Z 470.976,A -85,B 0,C 180,E1 11848.463,E2 11848.463} C_VEL
LIN {X 0,Y 343.916,Z 477.573,A -85,B 0,C 180,E1 11848.448,E2 11848.448} C_VEL
LIN {X 0,Y 340.339,Z 520.36,A -85,B 0,C 180,E1 11847.637,E2 11847.637} C_VEL
LIN {X 0,Y 336.735,Z 544.704,A -85,B 0,C 180,E1 11846.991,E2 11846.991} C_VEL
LIN {X 0,Y 332.823,Z 563.339,A -85,B 0,C 180,E1 11846.312,E2 11846.312} C_VEL
LIN {X 0,Y 328.494,Z 580.347,A -85,B 0,C 180,E1 11845.517,E2 11845.517} C_VEL
LIN {X 0,Y 323.779,Z 596.204,A -85,B 0,C 180,E1 11844.604,E2 11844.604} C_VEL
LIN {X 0,Y 318.381,Z 612.064,A -85,B 0,C 180,E1 11843.501,E2 11843.501} C_VEL
LIN {X 0,Y 312.46,Z 627.503,A -85,B 0,C 180,E1 11842.214,E2 11842.214} C_VEL
LIN {X 0,Y 306.1,Z 642.48,A -85,B 0,C 180,E1 11840.72,E2 11840.72} C_VEL
LIN {X 0,Y 298.469,Z 658.838,A -85,B 0,C 180,E1 11838.763,E2 11838.763} C_VEL
LIN {X 0,Y 289.268,Z 676.667,A -85,B 0,C 180,E1 11836.104,E2 11836.104} C_VEL
LIN {X 0,Y 282.012,Z 689.664,A -85,B 0,C 180,E1 11833.732,E2 11833.732} C_VEL
LIN {X 0,Y 275.028,Z 701.55,A -85,B 0,C 180,E1 11831.144,E2 11831.144} C_VEL
LIN {X 0,Y 268.625,Z 712.044,A -85,B 0,C 180,E1 11828.428,E2 11828.428} C_VEL
LIN {X 0,Y 262.442,Z 721.941,A -85,B 0,C 180,E1 11825.379,E2 11825.379} C_VEL
LIN {X 0,Y 256.668,Z 731.117,A -85,B 0,C 180,E1 11821.988,E2 11821.988} C_VEL
LIN {X 0,Y 250.951,Z 740.437,A -85,B 0,C 180,E1 11817.782,E2 11817.782} C_VEL
LIN {X 0,Y 245.897,Z 749.09,A -85,B 0,C 180,E1 11812.721,E2 11812.721} C_VEL
LIN {X 0,Y 242.999,Z 754.711,A -85,B 0,C 180,E1 11808.469,E2 11808.469} C_VEL
LIN {X 0,Y 241.227,Z 758.888,A -85,B 0,C 180,E1 11804.399,E2 11804.399} C_VEL
LIN {X 0,Y 240.282,Z 761.999,A -85,B 0,C 180,E1 11800.306,E2 11800.306} C_VEL
LIN {X 0,Y 239.978,Z 763.983,A -85,B 0,C 180,E1 11796.458,E2 11796.458} C_VEL
LIN {X 0,Y 239.965,Z 765.062,A -85,B 0,C 180,E1 11792.627,E2 11792.627} C_VEL
LIN {X 0,Y 239.985,Z 765.241,A -85,B 0,C 180,E1 11788.806,E2 11788.806} C_VEL
LIN {X 0,Y 239.948,Z 764.429,A -85,B 0,C 180,E1 11784.741,E2 11784.741} C_VEL
LIN {X 0,Y 240.165,Z 762.592,A -85,B 0,C 180,E1 11780.651,E2 11780.651} C_VEL
LIN {X 0,Y 241.007,Z 759.516,A -85,B 0,C 180,E1 11776.323,E2 11776.323} C_VEL
LIN {X 0,Y 242.675,Z 755.399,A -85,B 0,C 180,E1 11772.137,E2 11772.137} C_VEL
LIN {X 0,Y 245.16,Z 750.428,A -85,B 0,C 180,E1 11768.217,E2 11768.217} C_VEL
LIN {X 0,Y 248.675,Z 744.173,A -85,B 0,C 180,E1 11764.266,E2 11764.266} C_VEL
LIN {X 0,Y 253.204,Z 736.685,A -85,B 0,C 180,E1 11760.426,E2 11760.426} C_VEL
LIN {X 0,Y 259.822,Z 726.239,A -85,B 0,C 180,E1 11756.087,E2 11756.087} C_VEL
LIN {X 0,Y 267.329,Z 714.148,A -85,B 0,C 180,E1 11752.17,E2 11752.17} C_VEL
LIN {X 0,Y 274.078,Z 703.132,A -85,B 0,C 180,E1 11749.237,E2 11749.237} C_VEL
LIN {X 0,Y 280.467,Z 692.333,A -85,B 0,C 180,E1 11746.811,E2 11746.811} C_VEL
LIN {X 0,Y 287.482,Z 679.895,A -85,B 0,C 180,E1 11744.452,E2 11744.452} C_VEL
LIN {X 0,Y 294.362,Z 666.938,A -85,B 0,C 180,E1 11742.379,E2 11742.379} C_VEL
LIN {X 0,Y 301.171,Z 653.168,A -85,B 0,C 180,E1 11740.52,E2 11740.52} C_VEL
LIN {X 0,Y 308.304,Z 637.511,A -85,B 0,C 180,E1 11738.751,E2 11738.751} C_VEL
LIN {X 0,Y 316.648,Z 616.872,A -85,B 0,C 180,E1 11736.868,E2 11736.868} C_VEL
LIN {X 0,Y 322.757,Z 599.39,A -85,B 0,C 180,E1 11735.6,E2 11735.6} C_VEL
LIN {X 0,Y 327.905,Z 582.442,A -85,B 0,C 180,E1 11734.593,E2 11734.593} C_VEL
LIN {X 0,Y 332.288,Z 565.567,A -85,B 0,C 180,E1 11733.783,E2 11733.783} C_VEL
LIN {X 0,Y 336.05,Z 548.179,A -85,B 0,C 180,E1 11733.127,E2 11733.127} C_VEL
LIN {X 0,Y 339.209,Z 529.361,A -85,B 0,C 180,E1 11732.579,E2 11732.579} C_VEL
LIN {X 0,Y 341.999,Z 502.454,A -85,B 0,C 180,E1 11732.003,E2 11732.003} C_VEL
LIN {X 0,Y 352.509,Z 366.841,A -85,B 0,C 180,E1 11729.551,E2 11729.551} C_VEL
LIN {X 0,Y 345.936,Z 352.299,A -85,B 0,C 180,E1 11726.941,E2 11726.941} C_VEL
LIN {X 0,Y 340.222,Z 340.908,A -85,B 0,C 180,E1 11724.435,E2 11724.435} C_VEL
LIN {X 0,Y 333.691,Z 330.404,A -85,B 0,C 180,E1 11721.258,E2 11721.258} C_VEL
LIN {X 0,Y 329.19,Z 323.88,A -85,B 0,C 180,E1 11718.736,E2 11718.736} C_VEL
LIN {X 0,Y 326.729,Z 320.335,A -85,B 0,C 180,E1 11717.177,E2 11717.177} C_VEL
LIN {X 0,Y 323.855,Z 316.136,A -85,B 0,C 180,E1 11715.123,E2 11715.123} C_VEL
LIN {X 0,Y 320.676,Z 311.509,A -85,B 0,C 180,E1 11712.424,E2 11712.424} C_VEL
LIN {X 0,Y 317.857,Z 307.803,A -85,B 0,C 180,E1 11709.415,E2 11709.415} C_VEL
LIN {X 0,Y 317.103,Z 306.255,A -85,B 0,C 180,E1 11708.34,E2 11708.34} C_VEL
LIN {X 0,Y 314.095,Z 302.614,A -85,B 0,C 180,E1 11700.547,E2 11700.547} C_VEL
LIN {X 0,Y 314.217,Z 303.042,A -85,B 0,C 180,E1 11697.812,E2 11697.812} C_VEL
LIN {X 0,Y 317.333,Z 306.609,A -85,B 0,C 180,E1 11691.027,E2 11691.027} C_VEL
LIN {X 0,Y 319.788,Z 310.684,A -85,B 0,C 180,E1 11688.091,E2 11688.091} C_VEL
LIN {X 0,Y 321.211,Z 312.268,A -85,B 0,C 180,E1 11686.774,E2 11686.774} C_VEL
LIN {X 0,Y 325.09,Z 317.899,A -85,B 0,C 180,E1 11683.654,E2 11683.654} C_VEL
LIN {X 0,Y 328.805,Z 323.258,A -85,B 0,C 180,E1 11681.195,E2 11681.195} C_VEL
LIN {X 0,Y 333.717,Z 330.442,A -85,B 0,C 180,E1 11678.421,E2 11678.421} C_VEL
LIN {X 0,Y 341.597,Z 343.069,A -85,B 0,C 180,E1 11674.654,E2 11674.654} C_VEL
LIN {X 0,Y 349.466,Z 356.647,A -85,B 0,C 180,E1 11671.457,E2 11671.457} C_VEL
LIN {X 0,Y 360.163,Z 371.952,A -85,B 0,C 180,E1 11667.883,E2 11667.883} C_VEL
LIN {X 0,Y 374.038,Z 387.532,A -85,B 0,C 180,E1 11664.119,E2 11664.119} C_VEL
LIN {X 0,Y 396.678,Z 406.966,A -85,B 0,C 180,E1 11659.243,E2 11659.243} C_VEL
LIN {X 0,Y 407.221,Z 415.411,A -85,B 0,C 180,E1 11657.049,E2 11657.049} C_VEL
LIN {X 0,Y 415.659,Z 422.425,A -85,B 0,C 180,E1 11655.136,E2 11655.136} C_VEL
LIN {X 0,Y 424.57,Z 429.88,A -85,B 0,C 180,E1 11652.959,E2 11652.959} C_VEL
LIN {X 0,Y 432.151,Z 436.468,A -85,B 0,C 180,E1 11650.897,E2 11650.897} C_VEL
LIN {X 0,Y 440.893,Z 443.941,A -85,B 0,C 180,E1 11648.366,E2 11648.366} C_VEL
LIN {X 0,Y 450.05,Z 451.565,A -85,B 0,C 180,E1 11645.592,E2 11645.592} C_VEL
LIN {X 0,Y 457.596,Z 457.716,A -85,B 0,C 180,E1 11643.186,E2 11643.186} C_VEL
LIN {X 0,Y 465.011,Z 464.089,A -85,B 0,C 180,E1 11640.672,E2 11640.672} C_VEL
LIN {X 0,Y 470.656,Z 468.435,A -85,B 0,C 180,E1 11638.669,E2 11638.669} C_VEL
LIN {X 0,Y 476.826,Z 473.493,A -85,B 0,C 180,E1 11636.324,E2 11636.324} C_VEL
LIN {X 0,Y 481.537,Z 476.973,A -85,B 0,C 180,E1 11634.403,E2 11634.403} C_VEL
LIN {X 0,Y 486.833,Z 481.467,A -85,B 0,C 180,E1 11632.074,E2 11632.074} C_VEL
LIN {X 0,Y 491.759,Z 484.698,A -85,B 0,C 180,E1 11629.709,E2 11629.709} C_VEL
LIN {X 0,Y 496.275,Z 488.778,A -85,B 0,C 180,E1 11627.226,E2 11627.226} C_VEL
LIN {X 0,Y 500.208,Z 491.669,A -85,B 0,C 180,E1 11624.823,E2 11624.823} C_VEL
LIN {X 0,Y 503.633,Z 493.587,A -85,B 0,C 180,E1 11622.366,E2 11622.366} C_VEL
LIN {X 0,Y 505.101,Z 494.453,A -85,B 0,C 180,E1 11621.185,E2 11621.185} C_VEL
LIN {X 0,Y 507.31,Z 496.837,A -85,B 0,C 180,E1 11618.957,E2 11618.957} C_VEL
LIN {X 0,Y 509.298,Z 498.693,A -85,B 0,C 180,E1 11616.424,E2 11616.424} C_VEL
LIN {X 0,Y 510.55,Z 499.687,A -85,B 0,C 180,E1 11614.042,E2 11614.042} C_VEL
LIN {X 0,Y 511.333,Z 500.211,A -85,B 0,C 180,E1 11611.456,E2 11611.456} C_VEL
LIN {X 0,Y 511.347,Z 500.223,A -85,B 0,C 180,E1 11608.992,E2 11608.992} C_VEL
LIN {X 0,Y 510.773,Z 499.837,A -85,B 0,C 180,E1 11606.409,E2 11606.409} C_VEL
LIN {X 0,Y 509.483,Z 498.858,A -85,B 0,C 180,E1 11603.917,E2 11603.917} C_VEL
LIN {X 0,Y 507.652,Z 497.135,A -85,B 0,C 180,E1 11601.392,E2 11601.392} C_VEL
LIN {X 0,Y 505.459,Z 494.914,A -85,B 0,C 180,E1 11599.17,E2 11599.17} C_VEL
LIN {X 0,Y 504.263,Z 493.846,A -85,B 0,C 180,E1 11598.101,E2 11598.101} C_VEL
LIN {X 0,Y 500.926,Z 492.112,A -85,B 0,C 180,E1 11595.672,E2 11595.672} C_VEL
LIN {X 0,Y 496.931,Z 489.318,A -85,B 0,C 180,E1 11593.16,E2 11593.16} C_VEL
LIN {X 0,Y 492.795,Z 485.554,A -85,B 0,C 180,E1 11590.813,E2 11590.813} C_VEL
LIN {X 0,Y 487.41,Z 481.909,A -85,B 0,C 180,E1 11588.207,E2 11588.207} C_VEL
LIN {X 0,Y 482.057,Z 477.458,A -85,B 0,C 180,E1 11585.82,E2 11585.82} C_VEL
LIN {X 0,Y 478.568,Z 474.73,A -85,B 0,C 180,E1 11584.378,E2 11584.378} C_VEL
LIN {X 0,Y 472.359,Z 469.957,A -85,B 0,C 180,E1 11581.971,E2 11581.971} C_VEL
LIN {X 0,Y 467.413,Z 465.863,A -85,B 0,C 180,E1 11580.164,E2 11580.164} C_VEL
LIN {X 0,Y 460.532,Z 460.341,A -85,B 0,C 180,E1 11577.796,E2 11577.796} C_VEL
LIN {X 0,Y 453.822,Z 454.811,A -85,B 0,C 180,E1 11575.601,E2 11575.601} C_VEL
LIN {X 0,Y 445.564,Z 447.835,A -85,B 0,C 180,E1 11573.025,E2 11573.025} C_VEL
LIN {X 0,Y 436,Z 439.684,A -85,B 0,C 180,E1 11570.199,E2 11570.199} C_VEL
LIN {X 0,Y 428.094,Z 432.714,A -85,B 0,C 180,E1 11567.966,E2 11567.966} C_VEL
LIN {X 0,Y 420.046,Z 426.058,A -85,B 0,C 180,E1 11565.914,E2 11565.914} C_VEL
LIN {X 0,Y 410.08,Z 417.819,A -85,B 0,C 180,E1 11563.585,E2 11563.585} C_VEL
LIN {X 0,Y 400.722,Z 410.321,A -85,B 0,C 180,E1 11561.585,E2 11561.585} C_VEL
LIN {X 0,Y 384.233,Z 396.846,A -85,B 0,C 180,E1 11558.221,E2 11558.221} C_VEL
LIN {X 0,Y 368.969,Z 382.205,A -85,B 0,C 180,E1 11554.593,E2 11554.593} C_VEL
LIN {X 0,Y 356.044,Z 366.611,A -85,B 0,C 180,E1 11550.832,E2 11550.832} C_VEL
LIN {X 0,Y 341.237,Z 342.484,A -85,B 0,C 180,E1 11545.189,E2 11545.189} C_VEL
LIN {X 0,Y 333.638,Z 330.338,A -85,B 0,C 180,E1 11541.538,E2 11541.538} C_VEL
LIN {X 0,Y 327.747,Z 321.55,A -85,B 0,C 180,E1 11538.13,E2 11538.13} C_VEL
LIN {X 0,Y 323.813,Z 316.098,A -85,B 0,C 180,E1 11535.4,E2 11535.4} C_VEL
LIN {X 0,Y 320.541,Z 311.398,A -85,B 0,C 180,E1 11532.613,E2 11532.613} C_VEL
LIN {X 0,Y 317.764,Z 307.641,A -85,B 0,C 180,E1 11529.6,E2 11529.6} C_VEL
LIN {X 0,Y 317.144,Z 306.304,A -85,B 0,C 180,E1 11528.704,E2 11528.704} C_VEL
LIN {X 0,Y 314.092,Z 302.582,A -85,B 0,C 180,E1 11520.73,E2 11520.73} C_VEL
LIN {X 0,Y 314.266,Z 303.171,A -85,B 0,C 180,E1 11517.812,E2 11517.812} C_VEL
LIN {X 0,Y 317.357,Z 306.645,A -85,B 0,C 180,E1 11511.302,E2 11511.302} C_VEL
LIN {X 0,Y 319.732,Z 310.613,A -85,B 0,C 180,E1 11508.454,E2 11508.454} C_VEL
LIN {X 0,Y 321.244,Z 312.332,A -85,B 0,C 180,E1 11507.05,E2 11507.05} C_VEL
LIN {X 0,Y 325.016,Z 317.768,A -85,B 0,C 180,E1 11504.017,E2 11504.017} C_VEL
LIN {X 0,Y 328.848,Z 323.358,A -85,B 0,C 180,E1 11501.473,E2 11501.473} C_VEL
LIN {X 0,Y 332.679,Z 329.006,A -85,B 0,C 180,E1 11499.273,E2 11499.273} C_VEL
LIN {X 0,Y 338.403,Z 337.954,A -85,B 0,C 180,E1 11496.399,E2 11496.399} C_VEL
LIN {X 0,Y 341.877,Z 344.045,A -85,B 0,C 180,E1 11494.815,E2 11494.815} C_VEL
LIN {X 0,Y 347.144,Z 354.909,A -85,B 0,C 180,E1 11492.558,E2 11492.558} C_VEL
LIN {X 0,Y 352.552,Z 367.136,A -85,B 0,C 180,E1 11490.425,E2 11490.425} C_VEL
LIN {X 0,Y 343.916,Z 477.573,A -85,B 0,C 180,E1 11488.448,E2 11488.448} C_VEL
LIN {X 0,Y 342.824,Z 485.26,A -85,B 0,C 180,E1 11488.45,E2 11488.45} C_VEL
LIN {X 0,Y 337.957,Z 505.707,A -85,B 0,C 180,E1 11488.981,E2 11488.981} C_VEL
LIN {X 0,Y 336.945,Z 512.289,A -85,B 0,C 180,E1 11488.959,E2 11488.959} C_VEL
LIN {X 0,Y 334.574,Z 531.693,A -85,B 0,C 180,E1 11488.511,E2 11488.511} C_VEL
LIN {X 0,Y 331.506,Z 549.148,A -85,B 0,C 180,E1 11487.995,E2 11487.995} C_VEL
LIN {X 0,Y 327.71,Z 566.136,A -85,B 0,C 180,E1 11487.352,E2 11487.352} C_VEL
LIN {X 0,Y 323.053,Z 583.51,A -85,B 0,C 180,E1 11486.514,E2 11486.514} C_VEL
LIN {X 0,Y 317.098,Z 602.399,A -85,B 0,C 180,E1 11485.375,E2 11485.375} C_VEL
LIN {X 0,Y 309.245,Z 623.298,A -85,B 0,C 180,E1 11483.765,E2 11483.765} C_VEL
LIN {X 0,Y 302.332,Z 639.461,A -85,B 0,C 180,E1 11482.216,E2 11482.216} C_VEL
LIN {X 0,Y 295.658,Z 653.621,A -85,B 0,C 180,E1 11480.593,E2 11480.593} C_VEL
LIN {X 0,Y 288.654,Z 667.321,A -85,B 0,C 180,E1 11478.727,E2 11478.727} C_VEL
LIN {X 0,Y 281.53,Z 680.278,A -85,B 0,C 180,E1 11476.63,E2 11476.63} C_VEL
LIN {X 0,Y 274.057,Z 693.045,A -85,B 0,C 180,E1 11474.168,E2 11474.168} C_VEL
LIN {X 0,Y 265.064,Z 707.656,A -85,B 0,C 180,E1 11470.731,E2 11470.731} C_VEL
LIN {X 0,Y 257.059,Z 719.899,A -85,B 0,C 180,E1 11467.072,E2 11467.072} C_VEL
LIN {X 0,Y 250.838,Z 729.314,A -85,B 0,C 180,E1 11463.642,E2 11463.642} C_VEL
LIN {X 0,Y 245.505,Z 737.445,A -85,B 0,C 180,E1 11460.058,E2 11460.058} C_VEL
LIN {X 0,Y 241.088,Z 744.395,A -85,B 0,C 180,E1 11456.341,E2 11456.341} C_VEL
LIN {X 0,Y 237.41,Z 750.584,A -85,B 0,C 180,E1 11452.272,E2 11452.272} C_VEL
LIN {X 0,Y 234.622,Z 755.888,A -85,B 0,C 180,E1 11447.866,E2 11447.866} C_VEL
LIN {X 0,Y 232.667,Z 760.776,A -85,B 0,C 180,E1 11442.406,E2 11442.406} C_VEL
LIN {X 0,Y 231.998,Z 763.628,A -85,B 0,C 180,E1 11437.179,E2 11437.179} C_VEL
LIN {X 0,Y 231.962,Z 764.857,A -85,B 0,C 180,E1 11432.965,E2 11432.965} C_VEL
LIN {X 0,Y 231.989,Z 765.095,A -85,B 0,C 180,E1 11429.012,E2 11429.012} C_VEL
LIN {X 0,Y 231.951,Z 764.254,A -85,B 0,C 180,E1 11424.559,E2 11424.559} C_VEL
LIN {X 0,Y 232.195,Z 762.418,A -85,B 0,C 180,E1 11420.333,E2 11420.333} C_VEL
LIN {X 0,Y 233.126,Z 759.339,A -85,B 0,C 180,E1 11415.851,E2 11415.851} C_VEL
LIN {X 0,Y 234.876,Z 755.346,A -85,B 0,C 180,E1 11411.64,E2 11411.64} C_VEL
LIN {X 0,Y 237.597,Z 750.25,A -85,B 0,C 180,E1 11407.486,E2 11407.486} C_VEL
LIN {X 0,Y 241.336,Z 743.995,A -85,B 0,C 180,E1 11403.423,E2 11403.423} C_VEL
LIN {X 0,Y 246.123,Z 736.506,A -85,B 0,C 180,E1 11399.486,E2 11399.486} C_VEL
LIN {X 0,Y 253.076,Z 726.06,A -85,B 0,C 180,E1 11395.054,E2 11395.054} C_VEL
LIN {X 0,Y 260.927,Z 713.97,A -85,B 0,C 180,E1 11391.07,E2 11391.07} C_VEL
LIN {X 0,Y 267.953,Z 702.954,A -85,B 0,C 180,E1 11388.098,E2 11388.098} C_VEL
LIN {X 0,Y 274.585,Z 692.155,A -85,B 0,C 180,E1 11385.648,E2 11385.648} C_VEL
LIN {X 0,Y 281.696,Z 679.984,A -85,B 0,C 180,E1 11383.318,E2 11383.318} C_VEL
LIN {X 0,Y 288.833,Z 666.985,A -85,B 0,C 180,E1 11381.223,E2 11381.223} C_VEL
LIN {X 0,Y 295.972,Z 652.991,A -85,B 0,C 180,E1 11379.328,E2 11379.328} C_VEL
LIN {X 0,Y 303.309,Z 637.33,A -85,B 0,C 180,E1 11377.559,E2 11377.559} C_VEL
LIN {X 0,Y 311.951,Z 616.489,A -85,B 0,C 180,E1 11375.666,E2 11375.666} C_VEL
LIN {X 0,Y 318.137,Z 599.213,A -85,B 0,C 180,E1 11374.42,E2 11374.42} C_VEL
LIN {X 0,Y 323.408,Z 582.266,A -85,B 0,C 180,E1 11373.42,E2 11373.42} C_VEL
LIN {X 0,Y 327.891,Z 565.392,A -85,B 0,C 180,E1 11372.616,E2 11372.616} C_VEL
LIN {X 0,Y 331.733,Z 548.003,A -85,B 0,C 180,E1 11371.966,E2 11371.966} C_VEL
LIN {X 0,Y 334.959,Z 529.186,A -85,B 0,C 180,E1 11371.423,E2 11371.423} C_VEL
LIN {X 0,Y 337.818,Z 502.278,A -85,B 0,C 180,E1 11370.85,E2 11370.85} C_VEL
LIN {X 0,Y 348.284,Z 370.452,A -85,B 0,C 180,E1 11368.462,E2 11368.462} C_VEL
LIN {X 0,Y 342.116,Z 356.552,A -85,B 0,C 180,E1 11365.862,E2 11365.862} C_VEL
LIN {X 0,Y 337.211,Z 346.761,A -85,B 0,C 180,E1 11363.597,E2 11363.597} C_VEL
LIN {X 0,Y 331.225,Z 337.026,A -85,B 0,C 180,E1 11360.544,E2 11360.544} C_VEL
LIN {X 0,Y 326.013,Z 328.999,A -85,B 0,C 180,E1 11357.4,E2 11357.4} C_VEL
LIN {X 0,Y 322.308,Z 323.695,A -85,B 0,C 180,E1 11354.737,E2 11354.737} C_VEL
LIN {X 0,Y 319.32,Z 319.225,A -85,B 0,C 180,E1 11352.111,E2 11352.111} C_VEL
LIN {X 0,Y 316.535,Z 315.353,A -85,B 0,C 180,E1 11348.996,E2 11348.996} C_VEL
LIN {X 0,Y 315.865,Z 314.06,A -85,B 0,C 180,E1 11348.007,E2 11348.007} C_VEL
LIN {X 0,Y 313.111,Z 310.543,A -85,B 0,C 180,E1 11340.366,E2 11340.366} C_VEL
LIN {X 0,Y 313.265,Z 311.105,A -85,B 0,C 180,E1 11337.622,E2 11337.622} C_VEL
LIN {X 0,Y 316.154,Z 314.459,A -85,B 0,C 180,E1 11331.268,E2 11331.268} C_VEL
LIN {X 0,Y 318.637,Z 318.578,A -85,B 0,C 180,E1 11328.231,E2 11328.231} C_VEL
LIN {X 0,Y 319.84,Z 319.993,A -85,B 0,C 180,E1 11327.084,E2 11327.084} C_VEL
LIN {X 0,Y 323.624,Z 325.65,A -85,B 0,C 180,E1 11323.947,E2 11323.947} C_VEL
LIN {X 0,Y 327.131,Z 330.835,A -85,B 0,C 180,E1 11321.558,E2 11321.558} C_VEL
LIN {X 0,Y 331.783,Z 337.861,A -85,B 0,C 180,E1 11318.845,E2 11318.845} C_VEL
LIN {X 0,Y 339.232,Z 350.116,A -85,B 0,C 180,E1 11315.164,E2 11315.164} C_VEL
LIN {X 0,Y 347.03,Z 363.898,A -85,B 0,C 180,E1 11311.895,E2 11311.895} C_VEL
LIN {X 0,Y 357.574,Z 379.109,A -85,B 0,C 180,E1 11308.284,E2 11308.284} C_VEL
LIN {X 0,Y 371.159,Z 394.548,A -85,B 0,C 180,E1 11304.511,E2 11304.511} C_VEL
LIN {X 0,Y 393.792,Z 414.119,A -85,B 0,C 180,E1 11299.553,E2 11299.553} C_VEL
LIN {X 0,Y 404.512,Z 422.603,A -85,B 0,C 180,E1 11297.368,E2 11297.368} C_VEL
LIN {X 0,Y 413.862,Z 430.265,A -85,B 0,C 180,E1 11295.267,E2 11295.267} C_VEL
LIN {X 0,Y 422.941,Z 437.792,A -85,B 0,C 180,E1 11293.07,E2 11293.07} C_VEL
LIN {X 0,Y 431.549,Z 445.205,A -85,B 0,C 180,E1 11290.742,E2 11290.742} C_VEL
LIN {X 0,Y 439.384,Z 451.862,A -85,B 0,C 180,E1 11288.479,E2 11288.479} C_VEL
LIN {X 0,Y 448.672,Z 459.553,A -85,B 0,C 180,E1 11285.678,E2 11285.678} C_VEL
LIN {X 0,Y 456.91,Z 466.217,A -85,B 0,C 180,E1 11283.055,E2 11283.055} C_VEL
LIN {X 0,Y 463.906,Z 472.165,A -85,B 0,C 180,E1 11280.684,E2 11280.684} C_VEL
LIN {X 0,Y 469.373,Z 476.383,A -85,B 0,C 180,E1 11278.754,E2 11278.754} C_VEL
LIN {X 0,Y 475.568,Z 481.392,A -85,B 0,C 180,E1 11276.405,E2 11276.405} C_VEL
LIN {X 0,Y 480.241,Z 484.847,A -85,B 0,C 180,E1 11274.514,E2 11274.514} C_VEL
LIN {X 0,Y 485.698,Z 489.406,A -85,B 0,C 180,E1 11272.128,E2 11272.128} C_VEL
LIN {X 0,Y 490.727,Z 492.66,A -85,B 0,C 180,E1 11269.719,E2 11269.719} C_VEL
LIN {X 0,Y 495.226,Z 496.754,A -85,B 0,C 180,E1 11267.25,E2 11267.25} C_VEL
LIN {X 0,Y 499.165,Z 499.606,A -85,B 0,C 180,E1 11264.854,E2 11264.854} C_VEL
LIN {X 0,Y 502.75,Z 501.582,A -85,B 0,C 180,E1 11262.285,E2 11262.285} C_VEL
LIN {X 0,Y 504.086,Z 502.434,A -85,B 0,C 180,E1 11261.208,E2 11261.208} C_VEL
LIN {X 0,Y 506.307,Z 504.787,A -85,B 0,C 180,E1 11258.974,E2 11258.974} C_VEL
LIN {X 0,Y 508.313,Z 506.636,A -85,B 0,C 180,E1 11256.437,E2 11256.437} C_VEL
LIN {X 0,Y 509.568,Z 507.629,A -85,B 0,C 180,E1 11254.05,E2 11254.05} C_VEL
LIN {X 0,Y 510.357,Z 508.151,A -85,B 0,C 180,E1 11251.459,E2 11251.459} C_VEL
LIN {X 0,Y 510.37,Z 508.163,A -85,B 0,C 180,E1 11248.99,E2 11248.99} C_VEL
LIN {X 0,Y 509.79,Z 507.778,A -85,B 0,C 180,E1 11246.402,E2 11246.402} C_VEL
LIN {X 0,Y 508.563,Z 506.855,A -85,B 0,C 180,E1 11244.02,E2 11244.02} C_VEL
LIN {X 0,Y 506.764,Z 505.195,A -85,B 0,C 180,E1 11241.491,E2 11241.491} C_VEL
LIN {X 0,Y 504.444,Z 502.887,A -85,B 0,C 180,E1 11239.148,E2 11239.148} C_VEL
LIN {X 0,Y 503.241,Z 501.778,A -85,B 0,C 180,E1 11238.076,E2 11238.076} C_VEL
LIN {X 0,Y 499.891,Z 500.048,A -85,B 0,C 180,E1 11235.641,E2 11235.641} C_VEL
LIN {X 0,Y 495.859,Z 497.269,A -85,B 0,C 180,E1 11233.122,E2 11233.122} C_VEL
LIN {X 0,Y 491.577,Z 493.415,A -85,B 0,C 180,E1 11230.7,E2 11230.7} C_VEL
LIN {X 0,Y 485.848,Z 489.519,A -85,B 0,C 180,E1 11227.942,E2 11227.942} C_VEL
LIN {X 0,Y 480.518,Z 485.105,A -85,B 0,C 180,E1 11225.607,E2 11225.607} C_VEL
LIN {X 0,Y 476.582,Z 482.109,A -85,B 0,C 180,E1 11223.996,E2 11223.996} C_VEL
LIN {X 0,Y 470.409,Z 477.32,A -85,B 0,C 180,E1 11221.641,E2 11221.641} C_VEL
LIN {X 0,Y 465.679,Z 473.443,A -85,B 0,C 180,E1 11219.918,E2 11219.918} C_VEL
LIN {X 0,Y 458.669,Z 467.825,A -85,B 0,C 180,E1 11217.528,E2 11217.528} C_VEL
LIN {X 0,Y 450.111,Z 460.806,A -85,B 0,C 180,E1 11214.774,E2 11214.774} C_VEL
LIN {X 0,Y 442.793,Z 454.718,A -85,B 0,C 180,E1 11212.537,E2 11212.537} C_VEL
LIN {X 0,Y 433.178,Z 446.548,A -85,B 0,C 180,E1 11209.719,E2 11209.719} C_VEL
LIN {X 0,Y 423.928,Z 438.573,A -85,B 0,C 180,E1 11207.184,E2 11207.184} C_VEL
LIN {X 0,Y 415.02,Z 431.141,A -85,B 0,C 180,E1 11205.001,E2 11205.001} C_VEL
LIN {X 0,Y 407.093,Z 424.766,A -85,B 0,C 180,E1 11203.209,E2 11203.209} C_VEL
LIN {X 0,Y 395.856,Z 415.775,A -85,B 0,C 180,E1 11200.86,E2 11200.86} C_VEL
LIN {X 0,Y 371.82,Z 395.187,A -85,B 0,C 180,E1 11195.653,E2 11195.653} C_VEL
LIN {X 0,Y 358.036,Z 379.707,A -85,B 0,C 180,E1 11191.858,E2 11191.858} C_VEL
LIN {X 0,Y 347.327,Z 364.403,A -85,B 0,C 180,E1 11188.219,E2 11188.219} C_VEL
LIN {X 0,Y 339.406,Z 350.43,A -85,B 0,C 180,E1 11184.915,E2 11184.915} C_VEL
LIN {X 0,Y 332.847,Z 339.672,A -85,B 0,C 180,E1 11181.731,E2 11181.731} C_VEL
LIN {X 0,Y 328.081,Z 332.258,A -85,B 0,C 180,E1 11179.032,E2 11179.032} C_VEL
LIN {X 0,Y 325.19,Z 327.983,A -85,B 0,C 180,E1 11177.168,E2 11177.168} C_VEL
LIN {X 0,Y 322.268,Z 323.655,A -85,B 0,C 180,E1 11175.015,E2 11175.015} C_VEL
LIN {X 0,Y 319.19,Z 319.114,A -85,B 0,C 180,E1 11172.299,E2 11172.299} C_VEL
LIN {X 0,Y 316.448,Z 315.191,A -85,B 0,C 180,E1 11169.182,E2 11169.182} C_VEL
LIN {X 0,Y 315.904,Z 314.109,A -85,B 0,C 180,E1 11168.372,E2 11168.372} C_VEL
LIN {X 0,Y 313.11,Z 310.507,A -85,B 0,C 180,E1 11160.549,E2 11160.549} C_VEL
LIN {X 0,Y 313.353,Z 311.329,A -85,B 0,C 180,E1 11157.439,E2 11157.439} C_VEL
LIN {X 0,Y 316.177,Z 314.488,A -85,B 0,C 180,E1 11151.544,E2 11151.544} C_VEL
LIN {X 0,Y 318.581,Z 318.508,A -85,B 0,C 180,E1 11148.596,E2 11148.596} C_VEL
LIN {X 0,Y 319.871,Z 320.054,A -85,B 0,C 180,E1 11147.36,E2 11147.36} C_VEL
LIN {X 0,Y 323.436,Z 325.326,A -85,B 0,C 180,E1 11144.398,E2 11144.398} C_VEL
LIN {X 0,Y 327.306,Z 331.137,A -85,B 0,C 180,E1 11141.752,E2 11141.752} C_VEL
LIN {X 0,Y 331.76,Z 337.795,A -85,B 0,C 180,E1 11139.167,E2 11139.167} C_VEL
LIN {X 0,Y 338.23,Z 348.545,A -85,B 0,C 180,E1 11135.923,E2 11135.923} C_VEL
LIN {X 0,Y 343.724,Z 360.09,A -85,B 0,C 180,E1 11133.432,E2 11133.432} C_VEL
LIN {X 0,Y 348.345,Z 370.862,A -85,B 0,C 180,E1 11131.503,E2 11131.503} C_VEL
LIN {X 0,Y 336.945,Z 512.289,A -85,B 0,C 180,E1 11128.959,E2 11128.959} C_VEL
LIN {X 0,Y 335.611,Z 519.943,A -85,B 0,C 180,E1 11128.95,E2 11128.95} C_VEL
LIN {X 0,Y 329.119,Z 541.206,A -85,B 0,C 180,E1 11129.383,E2 11129.383} C_VEL
LIN {X 0,Y 327.814,Z 546.572,A -85,B 0,C 180,E1 11129.266,E2 11129.266} C_VEL
LIN {X 0,Y 323.82,Z 564.474,A -85,B 0,C 180,E1 11128.612,E2 11128.612} C_VEL
LIN {X 0,Y 319.401,Z 580.897,A -85,B 0,C 180,E1 11127.846,E2 11127.846} C_VEL
LIN {X 0,Y 314.369,Z 596.914,A -85,B 0,C 180,E1 11126.927,E2 11126.927} C_VEL
LIN {X 0,Y 308.638,Z 612.82,A -85,B 0,C 180,E1 11125.822,E2 11125.822} C_VEL
LIN {X 0,Y 302.15,Z 628.761,A -85,B 0,C 180,E1 11124.485,E2 11124.485} C_VEL
LIN {X 0,Y 293.509,Z 647.771,A -85,B 0,C 180,E1 11122.527,E2 11122.527} C_VEL
LIN {X 0,Y 284.597,Z 664.902,A -85,B 0,C 180,E1 11120.293,E2 11120.293} C_VEL
LIN {X 0,Y 277.06,Z 678.309,A -85,B 0,C 180,E1 11118.171,E2 11118.171} C_VEL
LIN {X 0,Y 269.922,Z 690.198,A -85,B 0,C 180,E1 11115.935,E2 11115.935} C_VEL
LIN {X 0,Y 262.571,Z 701.795,A -85,B 0,C 180,E1 11113.335,E2 11113.335} C_VEL
LIN {X 0,Y 255.56,Z 712.388,A -85,B 0,C 180,E1 11110.496,E2 11110.496} C_VEL
LIN {X 0,Y 248.456,Z 722.815,A -85,B 0,C 180,E1 11107.127,E2 11107.127} C_VEL
LIN {X 0,Y 240.81,Z 733.981,A -85,B 0,C 180,E1 11102.664,E2 11102.664} C_VEL
LIN {X 0,Y 234.594,Z 743.016,A -85,B 0,C 180,E1 11097.955,E2 11097.955} C_VEL
LIN {X 0,Y 230.41,Z 749.525,A -85,B 0,C 180,E1 11093.699,E2 11093.699} C_VEL
LIN {X 0,Y 227.448,Z 754.625,A -85,B 0,C 180,E1 11089.515,E2 11089.515} C_VEL
LIN {X 0,Y 225.435,Z 758.742,A -85,B 0,C 180,E1 11085.168,E2 11085.168} C_VEL
LIN {X 0,Y 224.344,Z 761.795,A -85,B 0,C 180,E1 11080.787,E2 11080.787} C_VEL
LIN {X 0,Y 223.983,Z 763.721,A -85,B 0,C 180,E1 11076.664,E2 11076.664} C_VEL
LIN {X 0,Y 223.969,Z 764.742,A -85,B 0,C 180,E1 11072.558,E2 11072.558} C_VEL
LIN {X 0,Y 223.988,Z 764.891,A -85,B 0,C 180,E1 11068.721,E2 11068.721} C_VEL
LIN {X 0,Y 223.956,Z 764.078,A -85,B 0,C 180,E1 11064.364,E2 11064.364} C_VEL
LIN {X 0,Y 224.267,Z 762.093,A -85,B 0,C 180,E1 11059.728,E2 11059.728} C_VEL
LIN {X 0,Y 225.26,Z 759.161,A -85,B 0,C 180,E1 11055.346,E2 11055.346} C_VEL
LIN {X 0,Y 227.158,Z 755.168,A -85,B 0,C 180,E1 11050.993,E2 11050.993} C_VEL
LIN {X 0,Y 230.074,Z 750.071,A -85,B 0,C 180,E1 11046.707,E2 11046.707} C_VEL
LIN {X 0,Y 234.053,Z 743.816,A -85,B 0,C 180,E1 11042.528,E2 11042.528} C_VEL
LIN {X 0,Y 239.112,Z 736.328,A -85,B 0,C 180,E1 11038.491,E2 11038.491} C_VEL
LIN {X 0,Y 246.418,Z 725.881,A -85,B 0,C 180,E1 11033.965,E2 11033.965} C_VEL
LIN {X 0,Y 254.626,Z 713.791,A -85,B 0,C 180,E1 11029.915,E2 11029.915} C_VEL
LIN {X 0,Y 261.938,Z 702.776,A -85,B 0,C 180,E1 11026.906,E2 11026.906} C_VEL
LIN {X 0,Y 269.37,Z 691.087,A -85,B 0,C 180,E1 11024.249,E2 11024.249} C_VEL
LIN {X 0,Y 277.06,Z 678.309,A -85,B 0,C 180,E1 11021.829,E2 11021.829} C_VEL
LIN {X 0,Y 284.908,Z 664.342,A -85,B 0,C 180,E1 11019.625,E2 11019.625} C_VEL
LIN {X 0,Y 294.483,Z 645.68,A -85,B 0,C 180,E1 11017.239,E2 11017.239} C_VEL
LIN {X 0,Y 302.15,Z 628.761,A -85,B 0,C 180,E1 11015.515,E2 11015.515} C_VEL
LIN {X 0,Y 308.644,Z 612.805,A -85,B 0,C 180,E1 11014.177,E2 11014.177} C_VEL
LIN {X 0,Y 314.369,Z 596.913,A -85,B 0,C 180,E1 11013.073,E2 11013.073} C_VEL
LIN {X 0,Y 319.406,Z 580.883,A -85,B 0,C 180,E1 11012.153,E2 11012.153} C_VEL
LIN {X 0,Y 323.82,Z 564.473,A -85,B 0,C 180,E1 11011.388,E2 11011.388} C_VEL
LIN {X 0,Y 327.814,Z 546.57,A -85,B 0,C 180,E1 11010.733,E2 11010.733} C_VEL
LIN {X 0,Y 331.608,Z 524.005,A -85,B 0,C 180,E1 11010.108,E2 11010.108} C_VEL
LIN {X 0,Y 334.81,Z 489.366,A -85,B 0,C 180,E1 11009.437,E2 11009.437} C_VEL
LIN {X 0,Y 344.231,Z 374.273,A -85,B 0,C 180,E1 11007.369,E2 11007.369} C_VEL
LIN {X 0,Y 338.492,Z 361.091,A -85,B 0,C 180,E1 11004.801,E2 11004.801} C_VEL
LIN {X 0,Y 334.437,Z 352.893,A -85,B 0,C 180,E1 11002.826,E2 11002.826} C_VEL
LIN {X 0,Y 328.598,Z 343.29,A -85,B 0,C 180,E1 10999.694,E2 10999.694} C_VEL
LIN {X 0,Y 323.997,Z 336.074,A -85,B 0,C 180,E1 10996.771,E2 10996.771} C_VEL
LIN {X 0,Y 320.666,Z 331.12,A -85,B 0,C 180,E1 10994.261,E2 10994.261} C_VEL
LIN {X 0,Y 317.974,Z 326.94,A -85,B 0,C 180,E1 10991.794,E2 10991.794} C_VEL
LIN {X 0,Y 315.231,Z 322.902,A -85,B 0,C 180,E1 10988.574,E2 10988.574} C_VEL
LIN {X 0,Y 314.637,Z 321.868,A -85,B 0,C 180,E1 10987.67,E2 10987.67} C_VEL
LIN {X 0,Y 312.136,Z 318.485,A -85,B 0,C 180,E1 10980.367,E2 10980.367} C_VEL
LIN {X 0,Y 312.287,Z 319.079,A -85,B 0,C 180,E1 10977.615,E2 10977.615} C_VEL
LIN {X 0,Y 314.981,Z 322.305,A -85,B 0,C 180,E1 10971.511,E2 10971.511} C_VEL
LIN {X 0,Y 317.488,Z 326.471,A -85,B 0,C 180,E1 10968.372,E2 10968.372} C_VEL
LIN {X 0,Y 318.566,Z 327.887,A -85,B 0,C 180,E1 10967.308,E2 10967.308} C_VEL
LIN {X 0,Y 322.054,Z 333.204,A -85,B 0,C 180,E1 10964.329,E2 10964.329} C_VEL
LIN {X 0,Y 325.601,Z 338.615,A -85,B 0,C 180,E1 10961.838,E2 10961.838} C_VEL
LIN {X 0,Y 329.941,Z 345.407,A -85,B 0,C 180,E1 10959.233,E2 10959.233} C_VEL
LIN {X 0,Y 336.811,Z 357.002,A -85,B 0,C 180,E1 10955.722,E2 10955.722} C_VEL
LIN {X 0,Y 352.413,Z 382.97,A -85,B 0,C 180,E1 10949.525,E2 10949.525} C_VEL
LIN {X 0,Y 367.261,Z 400.523,A -85,B 0,C 180,E1 10945.176,E2 10945.176} C_VEL
LIN {X 0,Y 389.983,Z 420.597,A -85,B 0,C 180,E1 10940.039,E2 10940.039} C_VEL
LIN {X 0,Y 400.53,Z 428.934,A -85,B 0,C 180,E1 10937.91,E2 10937.91} C_VEL
LIN {X 0,Y 410.827,Z 437.141,A -85,B 0,C 180,E1 10935.692,E2 10935.692} C_VEL
LIN {X 0,Y 420.398,Z 445.009,A -85,B 0,C 180,E1 10933.397,E2 10933.397} C_VEL
LIN {X 0,Y 428.292,Z 451.702,A -85,B 0,C 180,E1 10931.322,E2 10931.322} C_VEL
LIN {X 0,Y 436.826,Z 458.868,A -85,B 0,C 180,E1 10928.898,E2 10928.898} C_VEL
LIN {X 0,Y 446.622,Z 466.951,A -85,B 0,C 180,E1 10925.97,E2 10925.97} C_VEL
LIN {X 0,Y 454.41,Z 473.173,A -85,B 0,C 180,E1 10923.52,E2 10923.52} C_VEL
LIN {X 0,Y 461.711,Z 479.405,A -85,B 0,C 180,E1 10921.074,E2 10921.074} C_VEL
LIN {X 0,Y 468.009,Z 484.261,A -85,B 0,C 180,E1 10918.867,E2 10918.867} C_VEL
LIN {X 0,Y 474.345,Z 489.314,A -85,B 0,C 180,E1 10916.472,E2 10916.472} C_VEL
LIN {X 0,Y 478.986,Z 492.753,A -85,B 0,C 180,E1 10914.608,E2 10914.608} C_VEL
LIN {X 0,Y 484.39,Z 497.231,A -85,B 0,C 180,E1 10912.25,E2 10912.25} C_VEL
LIN {X 0,Y 489.509,Z 500.522,A -85,B 0,C 180,E1 10909.818,E2 10909.818} C_VEL
LIN {X 0,Y 494.204,Z 504.748,A -85,B 0,C 180,E1 10907.26,E2 10907.26} C_VEL
LIN {X 0,Y 498.119,Z 507.542,A -85,B 0,C 180,E1 10904.886,E2 10904.886} C_VEL
LIN {X 0,Y 501.728,Z 509.514,A -85,B 0,C 180,E1 10902.311,E2 10902.311} C_VEL
LIN {X 0,Y 503.071,Z 510.412,A -85,B 0,C 180,E1 10901.23,E2 10901.23} C_VEL
LIN {X 0,Y 505.303,Z 512.737,A -85,B 0,C 180,E1 10898.992,E2 10898.992} C_VEL
LIN {X 0,Y 507.271,Z 514.523,A -85,B 0,C 180,E1 10896.563,E2 10896.563} C_VEL
LIN {X 0,Y 508.586,Z 515.57,A -85,B 0,C 180,E1 10894.058,E2 10894.058} C_VEL
LIN {X 0,Y 509.381,Z 516.091,A -85,B 0,C 180,E1 10891.462,E2 10891.462} C_VEL
LIN {X 0,Y 509.394,Z 516.103,A -85,B 0,C 180,E1 10888.988,E2 10888.988} C_VEL
LIN {X 0,Y 508.808,Z 515.718,A -85,B 0,C 180,E1 10886.395,E2 10886.395} C_VEL
LIN {X 0,Y 507.577,Z 514.797,A -85,B 0,C 180,E1 10884.008,E2 10884.008} C_VEL
LIN {X 0,Y 505.759,Z 513.149,A -85,B 0,C 180,E1 10881.474,E2 10881.474} C_VEL
LIN {X 0,Y 503.429,Z 510.858,A -85,B 0,C 180,E1 10879.125,E2 10879.125} C_VEL
LIN {X 0,Y 502.049,Z 509.646,A -85,B 0,C 180,E1 10877.929,E2 10877.929} C_VEL
LIN {X 0,Y 498.688,Z 507.878,A -85,B 0,C 180,E1 10875.487,E2 10875.487} C_VEL
LIN {X 0,Y 494.787,Z 505.218,A -85,B 0,C 180,E1 10873.084,E2 10873.084} C_VEL
LIN {X 0,Y 490.539,Z 501.466,A -85,B 0,C 180,E1 10870.693,E2 10870.693} C_VEL
LIN {X 0,Y 484.863,Z 497.565,A -85,B 0,C 180,E1 10867.959,E2 10867.959} C_VEL
LIN {X 0,Y 479.5,Z 493.232,A -85,B 0,C 180,E1 10865.617,E2 10865.617} C_VEL
LIN {X 0,Y 475.563,Z 490.155,A -85,B 0,C 180,E1 10864.003,E2 10864.003} C_VEL
LIN {X 0,Y 469.32,Z 485.422,A -85,B 0,C 180,E1 10861.631,E2 10861.631} C_VEL
LIN {X 0,Y 463.912,Z 481.025,A -85,B 0,C 180,E1 10859.68,E2 10859.68} C_VEL
LIN {X 0,Y 456.839,Z 475.356,A -85,B 0,C 180,E1 10857.28,E2 10857.28} C_VEL
LIN {X 0,Y 448.187,Z 468.311,A -85,B 0,C 180,E1 10854.519,E2 10854.519} C_VEL
LIN {X 0,Y 440.633,Z 462.064,A -85,B 0,C 180,E1 10852.222,E2 10852.222} C_VEL
LIN {X 0,Y 430.814,Z 453.777,A -85,B 0,C 180,E1 10849.372,E2 10849.372} C_VEL
LIN {X 0,Y 422.422,Z 446.562,A -85,B 0,C 180,E1 10847.105,E2 10847.105} C_VEL
LIN {X 0,Y 414.109,Z 439.766,A -85,B 0,C 180,E1 10845.078,E2 10845.078} C_VEL
LIN {X 0,Y 404.665,Z 432.182,A -85,B 0,C 180,E1 10842.95,E2 10842.95} C_VEL
LIN {X 0,Y 393.701,Z 423.544,A -85,B 0,C 180,E1 10840.698,E2 10840.698} C_VEL
LIN {X 0,Y 368.82,Z 402.076,A -85,B 0,C 180,E1 10835.224,E2 10835.224} C_VEL
LIN {X 0,Y 355.116,Z 386.436,A -85,B 0,C 180,E1 10831.345,E2 10831.345} C_VEL
LIN {X 0,Y 344.518,Z 370.969,A -85,B 0,C 180,E1 10827.622,E2 10827.622} C_VEL
LIN {X 0,Y 336.811,Z 357.002,A -85,B 0,C 180,E1 10824.278,E2 10824.278} C_VEL
LIN {X 0,Y 329.651,Z 344.877,A -85,B 0,C 180,E1 10820.6,E2 10820.6} C_VEL
LIN {X 0,Y 324.34,Z 336.487,A -85,B 0,C 180,E1 10817.307,E2 10817.307} C_VEL
LIN {X 0,Y 320.63,Z 331.078,A -85,B 0,C 180,E1 10814.539,E2 10814.539} C_VEL
LIN {X 0,Y 317.849,Z 326.827,A -85,B 0,C 180,E1 10811.983,E2 10811.983} C_VEL
LIN {X 0,Y 315.149,Z 322.74,A -85,B 0,C 180,E1 10808.76,E2 10808.76} C_VEL
LIN {X 0,Y 314.551,Z 321.825,A -85,B 0,C 180,E1 10807.856,E2 10807.856} C_VEL
LIN {X 0,Y 312.135,Z 318.449,A -85,B 0,C 180,E1 10800.551,E2 10800.551} C_VEL
LIN {X 0,Y 312.375,Z 319.302,A -85,B 0,C 180,E1 10797.431,E2 10797.431} C_VEL
LIN {X 0,Y 315.003,Z 322.328,A -85,B 0,C 180,E1 10791.788,E2 10791.788} C_VEL
LIN {X 0,Y 317.431,Z 326.401,A -85,B 0,C 180,E1 10788.738,E2 10788.738} C_VEL
LIN {X 0,Y 318.508,Z 327.773,A -85,B 0,C 180,E1 10787.674,E2 10787.674} C_VEL
LIN {X 0,Y 321.981,Z 333.075,A -85,B 0,C 180,E1 10784.695,E2 10784.695} C_VEL
LIN {X 0,Y 325.57,Z 338.591,A -85,B 0,C 180,E1 10782.165,E2 10782.165} C_VEL
LIN {X 0,Y 329.844,Z 345.207,A -85,B 0,C 180,E1 10779.597,E2 10779.597} C_VEL
LIN {X 0,Y 335.83,Z 355.46,A -85,B 0,C 180,E1 10776.486,E2 10776.486} C_VEL
LIN {X 0,Y 340.951,Z 366.594,A -85,B 0,C 180,E1 10774.066,E2 10774.066} C_VEL
LIN {X 0,Y 344.266,Z 374.573,A -85,B 0,C 180,E1 10772.607,E2 10772.607} C_VEL
LIN {X 0,Y 332.283,Z 517.737,A -85,B 0,C 180,E1 10770.024,E2 10770.024} C_VEL
LIN {X 0,Y 329.369,Z 538.446,A -85,B 0,C 180,E1 10769.514,E2 10769.514} C_VEL
LIN {X 0,Y 327.814,Z 546.572,A -85,B 0,C 180,E1 10769.266,E2 10769.266} C_VEL
LIN {X 0,Y 325.724,Z 554.026,A -85,B 0,C 180,E1 10769.188,E2 10769.188} C_VEL
LIN {X 0,Y 317.667,Z 573.65,A -85,B 0,C 180,E1 10769.34,E2 10769.34} C_VEL
LIN {X 0,Y 315.468,Z 579.824,A -85,B 0,C 180,E1 10769.129,E2 10769.129} C_VEL
LIN {X 0,Y 310.413,Z 595.676,A -85,B 0,C 180,E1 10768.241,E2 10768.241} C_VEL
LIN {X 0,Y 304.611,Z 611.535,A -85,B 0,C 180,E1 10767.162,E2 10767.162} C_VEL
LIN {X 0,Y 298.226,Z 626.973,A -85,B 0,C 180,E1 10765.897,E2 10765.897} C_VEL
LIN {X 0,Y 291.339,Z 641.95,A -85,B 0,C 180,E1 10764.418,E2 10764.418} C_VEL
LIN {X 0,Y 283.35,Z 657.676,A -85,B 0,C 180,E1 10762.549,E2 10762.549} C_VEL
LIN {X 0,Y 272.924,Z 676.134,A -85,B 0,C 180,E1 10759.797,E2 10759.797} C_VEL
LIN {X 0,Y 264.896,Z 689.13,A -85,B 0,C 180,E1 10757.388,E2 10757.388} C_VEL
LIN {X 0,Y 257.105,Z 701.015,A -85,B 0,C 180,E1 10754.734,E2 10754.734} C_VEL
LIN {X 0,Y 249.808,Z 711.635,A -85,B 0,C 180,E1 10751.884,E2 10751.884} C_VEL
LIN {X 0,Y 242.87,Z 721.398,A -85,B 0,C 180,E1 10748.733,E2 10748.733} C_VEL
LIN {X 0,Y 236.216,Z 730.581,A -85,B 0,C 180,E1 10745.142,E2 10745.142} C_VEL
LIN {X 0,Y 229.529,Z 739.901,A -85,B 0,C 180,E1 10740.638,E2 10740.638} C_VEL
LIN {X 0,Y 223.492,Z 748.555,A -85,B 0,C 180,E1 10735.148,E2 10735.148} C_VEL
LIN {X 0,Y 219.942,Z 754.176,A -85,B 0,C 180,E1 10730.488,E2 10730.488} C_VEL
LIN {X 0,Y 217.704,Z 758.355,A -85,B 0,C 180,E1 10725.994,E2 10725.994} C_VEL
LIN {X 0,Y 216.448,Z 761.469,A -85,B 0,C 180,E1 10721.456,E2 10721.456} C_VEL
LIN {X 0,Y 215.999,Z 763.455,A -85,B 0,C 180,E1 10717.179,E2 10717.179} C_VEL
LIN {X 0,Y 215.965,Z 764.537,A -85,B 0,C 180,E1 10712.919,E2 10712.919} C_VEL
LIN {X 0,Y 215.988,Z 764.716,A -85,B 0,C 180,E1 10708.674,E2 10708.674} C_VEL
LIN {X 0,Y 215.962,Z 763.902,A -85,B 0,C 180,E1 10704.155,E2 10704.155} C_VEL
LIN {X 0,Y 216.317,Z 761.916,A -85,B 0,C 180,E1 10699.347,E2 10699.347} C_VEL
LIN {X 0,Y 217.413,Z 758.984,A -85,B 0,C 180,E1 10694.805,E2 10694.805} C_VEL
LIN {X 0,Y 219.47,Z 754.989,A -85,B 0,C 180,E1 10690.3,E2 10690.3} C_VEL
LIN {X 0,Y 222.596,Z 749.893,A -85,B 0,C 180,E1 10685.876,E2 10685.876} C_VEL
LIN {X 0,Y 226.83,Z 743.637,A -85,B 0,C 180,E1 10681.575,E2 10681.575} C_VEL
LIN {X 0,Y 232.178,Z 736.149,A -85,B 0,C 180,E1 10677.436,E2 10677.436} C_VEL
LIN {X 0,Y 240.057,Z 725.427,A -85,B 0,C 180,E1 10672.708,E2 10672.708} C_VEL
LIN {X 0,Y 248.434,Z 713.613,A -85,B 0,C 180,E1 10668.702,E2 10668.702} C_VEL
LIN {X 0,Y 256.042,Z 702.598,A -85,B 0,C 180,E1 10665.659,E2 10665.659} C_VEL
LIN {X 0,Y 263.751,Z 690.909,A -85,B 0,C 180,E1 10662.982,E2 10662.982} C_VEL
LIN {X 0,Y 271.704,Z 678.131,A -85,B 0,C 180,E1 10660.551,E2 10660.551} C_VEL
LIN {X 0,Y 279.802,Z 664.164,A -85,B 0,C 180,E1 10658.345,E2 10658.345} C_VEL
LIN {X 0,Y 289.655,Z 645.503,A -85,B 0,C 180,E1 10655.964,E2 10655.964} C_VEL
LIN {X 0,Y 297.741,Z 628.093,A -85,B 0,C 180,E1 10654.204,E2 10654.204} C_VEL
LIN {X 0,Y 304.254,Z 612.455,A -85,B 0,C 180,E1 10652.907,E2 10652.907} C_VEL
LIN {X 0,Y 310.048,Z 596.737,A -85,B 0,C 180,E1 10651.826,E2 10651.826} C_VEL
LIN {X 0,Y 315.212,Z 580.672,A -85,B 0,C 180,E1 10650.914,E2 10650.914} C_VEL
LIN {X 0,Y 319.711,Z 564.298,A -85,B 0,C 180,E1 10650.16,E2 10650.16} C_VEL
LIN {X 0,Y 323.788,Z 546.395,A -85,B 0,C 180,E1 10649.513,E2 10649.513} C_VEL
LIN {X 0,Y 327.658,Z 523.83,A -85,B 0,C 180,E1 10648.895,E2 10648.895} C_VEL
LIN {X 0,Y 330.943,Z 489.191,A -85,B 0,C 180,E1 10648.228,E2 10648.228} C_VEL
LIN {X 0,Y 340.256,Z 377.911,A -85,B 0,C 180,E1 10646.225,E2 10646.225} C_VEL
LIN {X 0,Y 334.66,Z 364.963,A -85,B 0,C 180,E1 10643.554,E2 10643.554} C_VEL
LIN {X 0,Y 331.714,Z 359.123,A -85,B 0,C 180,E1 10642.042,E2 10642.042} C_VEL
LIN {X 0,Y 326.252,Z 349.862,A -85,B 0,C 180,E1 10638.958,E2 10638.958} C_VEL
LIN {X 0,Y 321.903,Z 342.961,A -85,B 0,C 180,E1 10636.049,E2 10636.049} C_VEL
LIN {X 0,Y 319.153,Z 338.674,A -85,B 0,C 180,E1 10633.867,E2 10633.867} C_VEL
LIN {X 0,Y 316.459,Z 334.473,A -85,B 0,C 180,E1 10631.297,E2 10631.297} C_VEL
LIN {X 0,Y 313.889,Z 330.308,A -85,B 0,C 180,E1 10628.057,E2 10628.057} C_VEL
LIN {X 0,Y 313.073,Z 329.431,A -85,B 0,C 180,E1 10626.787,E2 10626.787} C_VEL
LIN {X 0,Y 311.161,Z 326.428,A -85,B 0,C 180,E1 10620.368,E2 10620.368} C_VEL
LIN {X 0,Y 311.309,Z 327.051,A -85,B 0,C 180,E1 10617.607,E2 10617.607} C_VEL
LIN {X 0,Y 313.814,Z 330.146,A -85,B 0,C 180,E1 10611.756,E2 10611.756} C_VEL
LIN {X 0,Y 316.341,Z 334.362,A -85,B 0,C 180,E1 10608.514,E2 10608.514} C_VEL
LIN {X 0,Y 317.385,Z 335.939,A -85,B 0,C 180,E1 10607.445,E2 10607.445} C_VEL
LIN {X 0,Y 320.5,Z 340.757,A -85,B 0,C 180,E1 10604.715,E2 10604.715} C_VEL
LIN {X 0,Y 323.889,Z 346.08,A -85,B 0,C 180,E1 10602.251,E2 10602.251} C_VEL
LIN {X 0,Y 328.116,Z 352.941,A -85,B 0,C 180,E1 10599.625,E2 10599.625} C_VEL
LIN {X 0,Y 334.504,Z 364.043,A -85,B 0,C 180,E1 10596.247,E2 10596.247} C_VEL
LIN {X 0,Y 349.57,Z 389.701,A -85,B 0,C 180,E1 10590.058,E2 10590.058} C_VEL
LIN {X 0,Y 364.176,Z 407.274,A -85,B 0,C 180,E1 10585.651,E2 10585.651} C_VEL
LIN {X 0,Y 386.78,Z 427.514,A -85,B 0,C 180,E1 10580.413,E2 10580.413} C_VEL
LIN {X 0,Y 398.873,Z 436.956,A -85,B 0,C 180,E1 10577.986,E2 10577.986} C_VEL
LIN {X 0,Y 408.681,Z 444.75,A -85,B 0,C 180,E1 10575.888,E2 10575.888} C_VEL
LIN {X 0,Y 418.368,Z 452.622,A -85,B 0,C 180,E1 10573.6,E2 10573.6} C_VEL
LIN {X 0,Y 426.979,Z 459.841,A -85,B 0,C 180,E1 10571.363,E2 10571.363} C_VEL
LIN {X 0,Y 435.065,Z 466.58,A -85,B 0,C 180,E1 10569.083,E2 10569.083} C_VEL
LIN {X 0,Y 444.665,Z 474.448,A -85,B 0,C 180,E1 10566.226,E2 10566.226} C_VEL
LIN {X 0,Y 452.446,Z 480.641,A -85,B 0,C 180,E1 10563.803,E2 10563.803} C_VEL
LIN {X 0,Y 460.023,Z 487.026,A -85,B 0,C 180,E1 10561.293,E2 10561.293} C_VEL
LIN {X 0,Y 466.296,Z 491.853,A -85,B 0,C 180,E1 10559.095,E2 10559.095} C_VEL
LIN {X 0,Y 472.686,Z 496.939,A -85,B 0,C 180,E1 10556.701,E2 10556.701} C_VEL
LIN {X 0,Y 477.707,Z 500.636,A -85,B 0,C 180,E1 10554.713,E2 10554.713} C_VEL
LIN {X 0,Y 483.182,Z 505.128,A -85,B 0,C 180,E1 10552.329,E2 10552.329} C_VEL
LIN {X 0,Y 488.663,Z 508.739,A -85,B 0,C 180,E1 10549.729,E2 10549.729} C_VEL
LIN {X 0,Y 493.278,Z 512.82,A -85,B 0,C 180,E1 10547.212,E2 10547.212} C_VEL
LIN {X 0,Y 497.338,Z 515.632,A -85,B 0,C 180,E1 10544.75,E2 10544.75} C_VEL
LIN {X 0,Y 500.866,Z 517.514,A -85,B 0,C 180,E1 10542.215,E2 10542.215} C_VEL
LIN {X 0,Y 502.258,Z 518.643,A -85,B 0,C 180,E1 10541.049,E2 10541.049} C_VEL
LIN {X 0,Y 504.523,Z 520.892,A -85,B 0,C 180,E1 10538.777,E2 10538.777} C_VEL
LIN {X 0,Y 506.463,Z 522.632,A -85,B 0,C 180,E1 10536.233,E2 10536.233} C_VEL
LIN {X 0,Y 507.711,Z 523.587,A -85,B 0,C 180,E1 10533.839,E2 10533.839} C_VEL
LIN {X 0,Y 508.412,Z 524.041,A -85,B 0,C 180,E1 10531.127,E2 10531.127} C_VEL
LIN {X 0,Y 508.407,Z 524.04,A -85,B 0,C 180,E1 10528.761,E2 10528.761} C_VEL
LIN {X 0,Y 507.711,Z 523.588,A -85,B 0,C 180,E1 10526.161,E2 10526.161} C_VEL
LIN {X 0,Y 506.462,Z 522.631,A -85,B 0,C 180,E1 10523.767,E2 10523.767} C_VEL
LIN {X 0,Y 504.523,Z 520.891,A -85,B 0,C 180,E1 10521.223,E2 10521.223} C_VEL
LIN {X 0,Y 502.259,Z 518.643,A -85,B 0,C 180,E1 10518.951,E2 10518.951} C_VEL
LIN {X 0,Y 500.866,Z 517.513,A -85,B 0,C 180,E1 10517.785,E2 10517.785} C_VEL
LIN {X 0,Y 497.338,Z 515.631,A -85,B 0,C 180,E1 10515.25,E2 10515.25} C_VEL
LIN {X 0,Y 493.278,Z 512.82,A -85,B 0,C 180,E1 10512.788,E2 10512.788} C_VEL
LIN {X 0,Y 488.652,Z 508.728,A -85,B 0,C 180,E1 10510.265,E2 10510.265} C_VEL
LIN {X 0,Y 483.182,Z 505.128,A -85,B 0,C 180,E1 10507.671,E2 10507.671} C_VEL
LIN {X 0,Y 477.707,Z 500.635,A -85,B 0,C 180,E1 10505.287,E2 10505.287} C_VEL
LIN {X 0,Y 472.693,Z 496.944,A -85,B 0,C 180,E1 10503.301,E2 10503.301} C_VEL
LIN {X 0,Y 466.196,Z 491.767,A -85,B 0,C 180,E1 10500.87,E2 10500.87} C_VEL
LIN {X 0,Y 459.306,Z 486.484,A -85,B 0,C 180,E1 10498.473,E2 10498.473} C_VEL
LIN {X 0,Y 450.859,Z 479.492,A -85,B 0,C 180,E1 10495.702,E2 10495.702} C_VEL
LIN {X 0,Y 442.876,Z 472.835,A -85,B 0,C 180,E1 10493.219,E2 10493.219} C_VEL
LIN {X 0,Y 433.916,Z 465.566,A -85,B 0,C 180,E1 10490.582,E2 10490.582} C_VEL
LIN {X 0,Y 424.476,Z 457.703,A -85,B 0,C 180,E1 10487.954,E2 10487.954} C_VEL
LIN {X 0,Y 416.003,Z 450.736,A -85,B 0,C 180,E1 10485.818,E2 10485.818} C_VEL
LIN {X 0,Y 406.892,Z 443.401,A -85,B 0,C 180,E1 10483.725,E2 10483.725} C_VEL
LIN {X 0,Y 396.236,Z 434.977,A -85,B 0,C 180,E1 10481.464,E2 10481.464} C_VEL
LIN {X 0,Y 370.716,Z 413.603,A -85,B 0,C 180,E1 10476.014,E2 10476.014} C_VEL
LIN {X 0,Y 357.293,Z 399.592,A -85,B 0,C 180,E1 10472.406,E2 10472.406} C_VEL
LIN {X 0,Y 345.594,Z 383.724,A -85,B 0,C 180,E1 10468.515,E2 10468.515} C_VEL
LIN {X 0,Y 333.843,Z 362.847,A -85,B 0,C 180,E1 10463.428,E2 10463.428} C_VEL
LIN {X 0,Y 327.405,Z 351.69,A -85,B 0,C 180,E1 10459.955,E2 10459.955} C_VEL
LIN {X 0,Y 322.475,Z 343.718,A -85,B 0,C 180,E1 10456.76,E2 10456.76} C_VEL
LIN {X 0,Y 319.014,Z 338.495,A -85,B 0,C 180,E1 10454.058,E2 10454.058} C_VEL
LIN {X 0,Y 316.518,Z 334.539,A -85,B 0,C 180,E1 10451.664,E2 10451.664} C_VEL
LIN {X 0,Y 313.922,Z 330.432,A -85,B 0,C 180,E1 10448.425,E2 10448.425} C_VEL
LIN {X 0,Y 313.34,Z 329.627,A -85,B 0,C 180,E1 10447.518,E2 10447.518} C_VEL
LIN {X 0,Y 311.159,Z 326.394,A -85,B 0,C 180,E1 10440.552,E2 10440.552} C_VEL
LIN {X 0,Y 311.397,Z 327.275,A -85,B 0,C 180,E1 10437.423,E2 10437.423} C_VEL
LIN {X 0,Y 313.835,Z 330.166,A -85,B 0,C 180,E1 10432.033,E2 10432.033} C_VEL
LIN {X 0,Y 316.284,Z 334.292,A -85,B 0,C 180,E1 10428.881,E2 10428.881} C_VEL
LIN {X 0,Y 317.414,Z 335.995,A -85,B 0,C 180,E1 10427.723,E2 10427.723} C_VEL
LIN {X 0,Y 320.427,Z 340.627,A -85,B 0,C 180,E1 10425.082,E2 10425.082} C_VEL
LIN {X 0,Y 323.926,Z 346.165,A -85,B 0,C 180,E1 10422.531,E2 10422.531} C_VEL
LIN {X 0,Y 328.019,Z 352.743,A -85,B 0,C 180,E1 10419.991,E2 10419.991} C_VEL
LIN {X 0,Y 333.384,Z 362.198,A -85,B 0,C 180,E1 10417.098,E2 10417.098} C_VEL
LIN {X 0,Y 338.179,Z 372.996,A -85,B 0,C 180,E1 10414.731,E2 10414.731} C_VEL
LIN {X 0,Y 340.309,Z 378.379,A -85,B 0,C 180,E1 10413.735,E2 10413.735} C_VEL
LIN {X 0,Y 328.35,Z 517.572,A -85,B 0,C 180,E1 10411.236,E2 10411.236} C_VEL
LIN {X 0,Y 325.328,Z 538.565,A -85,B 0,C 180,E1 10410.723,E2 10410.723} C_VEL
LIN {X 0,Y 320.477,Z 561.327,A -85,B 0,C 180,E1 10409.961,E2 10409.961} C_VEL
LIN {X 0,Y 315.587,Z 579.429,A -85,B 0,C 180,E1 10409.149,E2 10409.149} C_VEL
LIN {X 0,Y 315.468,Z 579.824,A -85,B 0,C 180,E1 10409.129,E2 10409.129} C_VEL
LIN {X 0,Y 312.731,Z 587.273,A -85,B 0,C 180,E1 10408.904,E2 10408.904} C_VEL
LIN {X 0,Y 303.386,Z 605.034,A -85,B 0,C 180,E1 10408.762,E2 10408.762} C_VEL
LIN {X 0,Y 300.203,Z 611.641,A -85,B 0,C 180,E1 10408.434,E2 10408.434} C_VEL
LIN {X 0,Y 293.774,Z 626.797,A -85,B 0,C 180,E1 10407.201,E2 10407.201} C_VEL
LIN {X 0,Y 286.707,Z 641.773,A -85,B 0,C 180,E1 10405.733,E2 10405.733} C_VEL
LIN {X 0,Y 278.496,Z 657.499,A -85,B 0,C 180,E1 10403.873,E2 10403.873} C_VEL
LIN {X 0,Y 267.924,Z 675.682,A -85,B 0,C 180,E1 10401.172,E2 10401.172} C_VEL
LIN {X 0,Y 259.452,Z 688.952,A -85,B 0,C 180,E1 10398.711,E2 10398.711} C_VEL
LIN {X 0,Y 251.377,Z 700.837,A -85,B 0,C 180,E1 10396.043,E2 10396.043} C_VEL
LIN {X 0,Y 243.882,Z 711.33,A -85,B 0,C 180,E1 10393.203,E2 10393.203} C_VEL
LIN {X 0,Y 236.548,Z 721.22,A -85,B 0,C 180,E1 10389.972,E2 10389.972} C_VEL
